# B&R Automation Studio project AutoCon2021 (part 3)

#### AngledMovementFb.st
```iecst
FUNCTION_BLOCK AngledMovementFb
	CASE Internal.state OF
		ANG_INT_OFF:
			IF Execute THEN
				Active := TRUE;
				Internal.ShPos[axPosX] := PosStartX - 0.026;
				Internal.ShPos[axPosY] := PosStartY + 0.026;
				Internal.ShPos[axPosZ] := 0.004;
				Internal.ShPos[axPosRX] := 0.025;
				Internal.ShPos[axPosRY] := 0.025;

				Internal.Fbs.Move6DFb.Controller := ADR(Controller);
				Internal.Fbs.Move6DFb.ShuttleID := ShuttleId;
				Internal.Fbs.Move6DFb.Position := Internal.ShPos;
				Internal.Fbs.Move6DFb.InPlaneVelocity := LinearVel;
				Internal.Fbs.Move6DFb.Acceleration := 10;
				Internal.Fbs.Move6DFb.ShortAxisVelocity[axVel] := LinearVel;
				Internal.Fbs.Move6DFb.ShortAxisVelocity[axVelRx] := ShortAxisRotVel;
				Internal.Fbs.Move6DFb.ShortAxisVelocity[axVelRy] := ShortAxisRotVel;
				Internal.Fbs.Move6DFb.ShortAxisVelocity[axVelRz] := ShortAxisRotVel;

				Internal.Fbs.Move6DFb.Execute := TRUE;

				Internal.state := ANG_INT_MOV_WAIT;
			END_IF
		ANG_INT_MOV_WAIT:
			IF Internal.Fbs.Move6DFb.Done THEN
				Internal.Fbs.Move6DFb.Execute := FALSE;
				Internal.MovementNum := Internal.MovementNum + 1;
				IF Internal.MovementNum >= 11 THEN
					Done := TRUE;
					Internal.state := ANG_INT_DONE;
				ELSE
					Internal.state := ANG_INT_MOV_WAIT + Internal.MovementNum;
				END_IF

			END_IF
		ANG_INT_MOV_1:
			Internal.ShPos[axPosX] := Internal.ShPos[axPosX];
			Internal.ShPos[axPosY] := Internal.ShPos[axPosY] - 0.052;
			Internal.ShPos[axPosRX] := -0.025;
			Internal.ShPos[axPosRY] := 0.025;

			Internal.Fbs.Move6DFb.Position := Internal.ShPos;
			Internal.Fbs.Move6DFb.Execute := TRUE;

			Internal.state := ANG_INT_MOV_WAIT;
		ANG_INT_MOV_2:
			Internal.ShPos[axPosX] := Internal.ShPos[axPosX] + 0.052;
			Internal.ShPos[axPosY] := Internal.ShPos[axPosY];
			Internal.ShPos[axPosRX] := -0.025;
			Internal.ShPos[axPosRY] := -0.025;

			Internal.Fbs.Move6DFb.Position := Internal.ShPos;
			Internal.Fbs.Move6DFb.Execute := TRUE;

			Internal.state := ANG_INT_MOV_WAIT;
		ANG_INT_MOV_3:
			Internal.ShPos[axPosX] := Internal.ShPos[axPosX];
			Internal.ShPos[axPosY] := Internal.ShPos[axPosY] + 0.052;
			Internal.ShPos[axPosRX] := 0.025;
			Internal.ShPos[axPosRY] := -0.025;

			Internal.Fbs.Move6DFb.Position := Internal.ShPos;
			Internal.Fbs.Move6DFb.Execute := TRUE;

			Internal.state := ANG_INT_MOV_WAIT;
		ANG_INT_MOV_4:
			Internal.ShPos[axPosX] := Internal.ShPos[axPosX] - 0.052;
			Internal.ShPos[axPosY] := Internal.ShPos[axPosY];
			Internal.ShPos[axPosRX] := 0.025;
			Internal.ShPos[axPosRY] := 0.025;

			Internal.Fbs.Move6DFb.Position := Internal.ShPos;
			Internal.Fbs.Move6DFb.Execute := TRUE;

			Internal.state := ANG_INT_MOV_WAIT;
		ANG_INT_MOV_5:
			Internal.ShPos[axPosX] := Internal.ShPos[axPosX] + 0.015;
			Internal.ShPos[axPosY] := Internal.ShPos[axPosY] - 0.015;
			Internal.ShPos[axPosRX] := 0.0;
			Internal.ShPos[axPosRY] := 0.0;

			Internal.Fbs.Move6DFb.Position := Internal.ShPos;
			Internal.Fbs.Move6DFb.Execute := TRUE;

			Internal.state := ANG_INT_MOV_WAIT;
		ANG_INT_MOV_6:
			Internal.ShPos[axPosX] := Internal.ShPos[axPosX];
			Internal.ShPos[axPosY] := Internal.ShPos[axPosY] - 0.026;
			Internal.ShPos[axPosRX] := 0.0;
			Internal.ShPos[axPosRY] := 0.0;

			Internal.Fbs.Move6DFb.Position := Internal.ShPos;
			Internal.Fbs.Move6DFb.Execute := TRUE;

			Internal.state := ANG_INT_MOV_WAIT;
		ANG_INT_MOV_7:
			Internal.ShPos[axPosX] := Internal.ShPos[axPosX] + 0.026;
			Internal.ShPos[axPosY] := Internal.ShPos[axPosY];
			Internal.ShPos[axPosRX] := 0.0;
			Internal.ShPos[axPosRY] := 0.0;

			Internal.Fbs.Move6DFb.Position := Internal.ShPos;
			Internal.Fbs.Move6DFb.Execute := TRUE;

			Internal.state := ANG_INT_MOV_WAIT;
		ANG_INT_MOV_8:
			Internal.ShPos[axPosX] := Internal.ShPos[axPosX];
			Internal.ShPos[axPosY] := Internal.ShPos[axPosY] + 0.026;
			Internal.ShPos[axPosRX] := 0.0;
			Internal.ShPos[axPosRY] := 0.0;

			Internal.Fbs.Move6DFb.Position := Internal.ShPos;
			Internal.Fbs.Move6DFb.Execute := TRUE;

			Internal.state := ANG_INT_MOV_WAIT;
		ANG_INT_MOV_9:
			Internal.ShPos[axPosX] := Internal.ShPos[axPosX] - 0.026;
			Internal.ShPos[axPosY] := Internal.ShPos[axPosY];
			Internal.ShPos[axPosRX] := 0.0;
			Internal.ShPos[axPosRY] := 0.0;

			Internal.Fbs.Move6DFb.Position := Internal.ShPos;
			Internal.Fbs.Move6DFb.Execute := TRUE;

			Internal.state := ANG_INT_MOV_WAIT;
		ANG_INT_MOV_10:
			Internal.ShPos[axPosX] := PosStartX;
			Internal.ShPos[axPosY] := PosStartY;
			Internal.ShPos[axPosZ] := 0.002;
			Internal.ShPos[axPosRX] := 0.0;
			Internal.ShPos[axPosRY] := 0.0;

			Internal.Fbs.Move6DFb.Position := Internal.ShPos;
			Internal.Fbs.Move6DFb.Execute := TRUE;

			Internal.state := ANG_INT_MOV_WAIT;

		ANG_INT_DONE:
			IF NOT Execute THEN
				Internal.Fbs.Move6DFb.Execute := FALSE;
				Internal.MovementNum := 0;

				Active := FALSE;
				Done := FALSE;
				Error := FALSE;

				Internal.state := ANG_INT_OFF;
			END_IF
		ANG_INT_ERROR:
			IF NOT Execute THEN
				Internal.Fbs.Move6DFb.Execute := FALSE;
				Internal.MovementNum := 0;

				Active := FALSE;
				Done := FALSE;
				Error := FALSE;

				Internal.state := ANG_INT_OFF;
			END_IF
	END_CASE;
	Internal.Fbs.Move6DFb();
END_FUNCTION_BLOCK
```

#### WobbleMovementFb.st
```iecst
FUNCTION_BLOCK WobbleMovementFb
	//Setup Sun/Planet
	//Run Macro on Virtual
	//Run Wobble Macro on Real
	//When Virtual macro finishes, issue stop command to Real
	//Move6D to real shuttle
	//Exit Sun/Planet
	CASE Internal.state OF
		WOB_INT_OFF:
			IF Execute THEN
				Active := TRUE;

				Internal.Fbs.PlanetCtrlFb.Controller := ADR(Controller);
				Internal.Fbs.PlanetCtrlFb.NumberOfPlanets := 1;
				Internal.Fbs.PlanetCtrlFb.PlanetShuttleID[0] := ShuttleId;
				Internal.Fbs.PlanetCtrlFb.StarShuttleID := VirtShId;
				Internal.Fbs.PlanetCtrlFb.Level := mcACP6D_PLANET_CONNECT;
				Internal.Fbs.PlanetCtrlFb.Execute := TRUE;

				Internal.state := WOB_INT_SETUP_PLANET;
			END_IF
		WOB_INT_SETUP_PLANET:
			IF Internal.Fbs.PlanetCtrlFb.Error THEN
				Internal.state := WOB_INT_ERROR;
			ELSIF Internal.Fbs.PlanetCtrlFb.Done THEN
				Internal.Fbs.PlanetCtrlFb.Execute := FALSE;

				Internal.Fbs.VirtualMacroFb.Controller := ADR(Controller);
				Internal.Fbs.VirtualMacroFb.MacroID := SunMacroID;
				Internal.Fbs.VirtualMacroFb.ShuttleID := VirtShId;
				Internal.Fbs.VirtualMacroFb.Execute := TRUE;

				Internal.Fbs.RealMacroFb.Controller := ADR(Controller);
				Internal.Fbs.RealMacroFb.MacroID := PlanetMacroID;
				Internal.Fbs.RealMacroFb.ShuttleID := ShuttleId;
				Internal.Fbs.RealMacroFb.Execute := TRUE;

				Internal.state := WOB_INT_MACRO_RUN;
			END_IF
		WOB_INT_MACRO_RUN:
			IF Internal.Fbs.RealMacroFb.Error OR Internal.Fbs.VirtualMacroFb.Error THEN
				Internal.state := WOB_INT_ERROR;
			ELSIF Internal.Fbs.VirtualMacroFb.Done THEN
				Internal.Fbs.VirtualMacroFb.Execute := FALSE;
				Internal.Fbs.RealMacroFb.Execute := FALSE;

				Internal.Fbs.StopFb.Controller := ADR(Controller);
				Internal.Fbs.StopFb.ShuttleID := ShuttleId;
				Internal.Fbs.StopFb.Execute := TRUE;

				Internal.state := WOB_INT_STOP;
			END_IF
		WOB_INT_STOP:
			IF Internal.Fbs.StopFb.Error THEN
				Internal.state := WOB_INT_ERROR;
			ELSIF Internal.Fbs.StopFb.Done THEN
				Internal.Fbs.StopFb.Execute := FALSE;

				Internal.Fbs.Move6DFb.Controller := ADR(Controller);
				Internal.Fbs.Move6DFb.ShuttleID := ShuttleId;
				Internal.Fbs.Move6DFb.Position[axPosX] := PosStartX;
				Internal.Fbs.Move6DFb.Position[axPosY] := PosStartY;
				Internal.Fbs.Move6DFb.Position[axPosZ] := 0.002;
				Internal.Fbs.Move6DFb.Position[axPosRX] := 0;
				Internal.Fbs.Move6DFb.Position[axPosRY] := 0;
				Internal.Fbs.Move6DFb.Position[axPosRZ] := 0;
				Internal.Fbs.Move6DFb.InPlaneVelocity := 1;
				Internal.Fbs.Move6DFb.Acceleration := 10;
				Internal.Fbs.Move6DFb.ShortAxisVelocity[axVel] := 1;
				Internal.Fbs.Move6DFb.ShortAxisVelocity[axVelRx] := 0.1;
				Internal.Fbs.Move6DFb.ShortAxisVelocity[axVelRy] := 0.1;
				Internal.Fbs.Move6DFb.ShortAxisVelocity[axVelRz] := 0.1;
				Internal.Fbs.Move6DFb.Execute := TRUE;

				Internal.state := WOB_INT_REORIENT;
			END_IF
		WOB_INT_REORIENT:
			IF Internal.Fbs.Move6DFb.Done THEN
				Internal.Fbs.Move6DFb.Execute := FALSE;

				Internal.Fbs.PlanetCtrlFb.Level := mcACP6D_PLANET_DISCONNECT;
				Internal.Fbs.PlanetCtrlFb.Execute := TRUE;

				Internal.state := WOB_INT_BREAK_PLANET;
			END_IF
		WOB_INT_BREAK_PLANET:
			IF Internal.Fbs.PlanetCtrlFb.Error THEN
				Internal.state := WOB_INT_ERROR;
			ELSIF Internal.Fbs.PlanetCtrlFb.Done THEN
				Internal.Fbs.PlanetCtrlFb.Execute := FALSE;
				Done := TRUE;

				Internal.state := WOB_INT_DONE;
			END_IF
		WOB_INT_DONE:
			IF NOT Execute THEN

				Active := FALSE;
				Done := FALSE;
				Error := FALSE;

				Internal.state := WOB_INT_OFF;
			END_IF
		WOB_INT_ERROR:
			IF NOT Execute THEN
				Internal.Fbs.PlanetCtrlFb.Execute := FALSE;
				Internal.Fbs.RealMacroFb.Execute := FALSE;
				Internal.Fbs.VirtualMacroFb.Execute := FALSE;
				Internal.Fbs.StopFb.Execute := FALSE;
				Internal.Fbs.Move6DFb.Execute := FALSE;

				Active := FALSE;
				Done := FALSE;
				Error := FALSE;

				Internal.state := WOB_INT_OFF;
			END_IF
	END_CASE;
	Internal.Fbs.PlanetCtrlFb();
	Internal.Fbs.RealMacroFb();
	Internal.Fbs.VirtualMacroFb();
	Internal.Fbs.StopFb();
	Internal.Fbs.Move6DFb();
END_FUNCTION_BLOCK
```

#### StationActions.st
```iecst
ACTION SetupStationActions:
	CASE station OF
		ST1:
			FillStationFbs.St1Fb.Execute := TRUE;
			FillStationFbs.St1Fb.Controller := ADR(gMcAcp6DController);
			FillStationFbs.St1Fb.ShuttleId := gShuttleIf[pFillIf.Par.ShuttleIdx].Cfg.ShuttleId;
			FillStationFbs.St1Fb.PosStartX := pFillIf.Cfg.StationPos.X;
			FillStationFbs.St1Fb.PosStartY := pFillIf.Cfg.StationPos.Y;
		ST2:
			FillStationFbs.St2Fb.Controller := ADR(gMcAcp6DController);
			FillStationFbs.St2Fb.MacroID := DINT_TO_USINT(MACRO_FILL_STATION_PROC_2);
			FillStationFbs.St2Fb.ShuttleID := gShuttleIf[pFillIf.Par.ShuttleIdx].Cfg.ShuttleId;
			FillStationFbs.St2Fb.Execute := TRUE;
		ST3:
			FillStationFbs.St3Fb.Controller := ADR(gMcAcp6DController);
			FillStationFbs.St3Fb.PosStartX := pFillIf.Cfg.StationPos.X;
			FillStationFbs.St3Fb.PosStartY := pFillIf.Cfg.StationPos.Y;
			FillStationFbs.St3Fb.PlanetMacroID := DINT_TO_USINT(MACRO_FILL_STATION_PROC_3_WOBBLE);

			FillStationFbs.St3Fb.ShuttleId := gShuttleIf[pFillIf.Par.ShuttleIdx].Cfg.ShuttleId;
			FillStationFbs.St3Fb.VirtShId := 100;
			FillStationFbs.St3Fb.Execute := TRUE;

			CASE macroPatternCounter OF
				0:
					FillStationFbs.St3Fb.SunMacroID := DINT_TO_USINT(MACRO_FILL_STATION_PROC_3_XY);
				1:
					FillStationFbs.St3Fb.SunMacroID := DINT_TO_USINT(MACRO_FILL_STATION_PROC_3_A);
				2:
					FillStationFbs.St3Fb.SunMacroID := DINT_TO_USINT(MACRO_FILL_STATION_PROC_3_B);
			END_CASE;

		ST4:
			FillStationFbs.St4Fb.Controller := ADR(gMcAcp6DController);
			FillStationFbs.St4Fb.MacroID := DINT_TO_USINT(MACRO_FILL_STATION_PROC_4);
			FillStationFbs.St4Fb.ShuttleID := gShuttleIf[pFillIf.Par.ShuttleIdx].Cfg.ShuttleId;
			FillStationFbs.St4Fb.Execute := TRUE;
	END_CASE;
END_ACTION

ACTION CallStationFbs:
	CASE station OF
		ST1:
			FillStationFbs.St1Fb();
		ST2:
			FillStationFbs.St2Fb();
		ST3:
			FillStationFbs.St3Fb();
		ST4:
			FillStationFbs.St4Fb();
	END_CASE;
END_ACTION
```

### Program Logical/Source/ProcessStations/FinishStation (IEC)

#### Cyclic.st - Cyclic code
```iecst
PROGRAM _CYCLIC
	//System operates a batching setup
	//Need two seperate state machines
	//One controls the ouside interface, basically the same as before

	//Second is the internal one, communicates to the external interface as well
	//Process

	//External state machine
	//Waits for a shuttle to be ready
	//When a shuttle is commanded to process
	//Inform the internal state machine a shuttle has arrived
	//Wait for acknowledge, go back to the Wait state

	//FB perhaps?
	//Internal state machine
	//Wait for a shuttle command
	//Send that shuttle to the appropriate destination
		// If the shuttle count is = # of stations, wait for the move to be done
			//Preform the process
		//Else
			//Head back to wait for a more shuttles

	IF NOT gFinishStationIf.Cmd.LocalOverride THEN
		stationPars := gSysPars.FinishStation;
	END_IF

	CASE state OF
		FINISH_OFF: //********************************************************************************Finish station is currently disabled
			IF gFinishStationIf.Cmd.Enable THEN
				stationFbs.BatchProcessFb.Controller := ADR(gMcAcp6DController);
				stationFbs.BatchProcessFb.Enable := TRUE;

				state := FINISH_INIT;
			END_IF
		FINISH_INIT: //********************************************************************************Finish station is initalizing
			IF stationFbs.BatchProcessFb.ReadyForShuttle THEN
				gFinishStationIf.Sts.ReadyForNewShuttle := TRUE;
				gFinishStationIf.Sts.Enabled := TRUE;
				state := FINISH_WAIT_FOR_SHUTTLE;
			END_IF
		FINISH_WAIT_FOR_SHUTTLE: //********************************************************************************Finish station is waiting for a shuttle to be present
			stationFbs.BatchProcessFb.ProcessingTime := stationPars.WaitTime;
			IF NOT gFinishStationIf.Cmd.Enable THEN
				gFinishStationIf.Sts.ReadyForNewShuttle := FALSE;
				gFinishStationIf.Sts.Enabled := FALSE;
				state := FINISH_OFF;
			ELSIF gFinishStationIf.Par.ShuttleIdx <> STATION_IS_EMPTY AND gFinishStationIf.Cmd.Process THEN
				gFinishStationIf.Sts.ReadyForNewShuttle := FALSE;

				stationFbs.BatchProcessFb.ShId := gShuttleIf[gFinishStationIf.Par.ShuttleIdx].Cfg.ShuttleId;
				stationFbs.BatchProcessFb.ProcessShuttle := TRUE;

				state := FINISH_CHECK_BUFFER;
			END_IF
		FINISH_CHECK_BUFFER:
			IF stationFbs.BatchProcessFb.Processsing THEN
				gFinishStationIf.Sts.Processing := TRUE;
				gFinishStationIf.Par.ShuttleIdx := STATION_IS_EMPTY;
				stationFbs.BatchProcessFb.ProcessShuttle := FALSE;

				state := FINISH_FINISHING;
			ELSIF stationFbs.BatchProcessFb.ReadyForShuttle THEN
				gFinishStationIf.Sts.ReadyForNewShuttle := TRUE;
				gFinishStationIf.Par.ShuttleIdx := STATION_IS_EMPTY;
				stationFbs.BatchProcessFb.ProcessShuttle := FALSE;

				state := FINISH_WAIT_FOR_SHUTTLE;
			END_IF
		FINISH_FINISHING: //********************************************************************************Finish station is loading product onto a shuttle
			IF stationFbs.BatchProcessFb.Error THEN
				gFinishStationIf.Sts.Error := TRUE;
				state := FINISH_ERROR;
			ELSIF stationFbs.BatchProcessFb.BatchComplete THEN
				stationFbs.BatchProcessFb.Reset := TRUE;
				gFinishStationIf.Cmd.Process := FALSE;

				gFinishStationIf.Sts.Processing := FALSE;
				FOR i:=0 TO MAX_BATCH_SHUTTLE_COUNT -1 DO
					gShuttleIf[stationFbs.BatchProcessFb.ShuttleIds[i] - 1].Cmd.NextStep := TRUE; //WARNING WARNING THIS WILL ONLY WORK WITH SEQUENTIAL IDS. IF YOU USE ABSOLUTE ID THIS WILL NOT WORK
					gShuttleIf[stationFbs.BatchProcessFb.ShuttleIds[i] - 1].Sts.ProductInfo.Finished := TRUE;
				END_FOR;

				gFinishStationIf.Sts.Done := TRUE;

				state := FINISH_DONE;
			END_IF
		FINISH_DONE: //********************************************************************************Finish station is done with the load process
			IF NOT gFinishStationIf.Cmd.Enable THEN
				gFinishStationIf.Sts.Done := FALSE;
				gFinishStationIf.Sts.Enabled := FALSE;
				gFinishStationIf.Sts.ReadyForNewShuttle := FALSE;
				stationFbs.BatchProcessFb.Enable := FALSE;

				state := FINISH_OFF;
			ELSIF NOT gFinishStationIf.Cmd.Process AND stationFbs.BatchProcessFb.ReadyForShuttle THEN
				gFinishStationIf.Par.ShuttleIdx := STATION_IS_EMPTY;
				gFinishStationIf.Sts.Done := FALSE;
				gFinishStationIf.Sts.ReadyForNewShuttle := FALSE;
				gFinishStationIf.Sts.ReadyForNewShuttle := TRUE;

				state := FINISH_WAIT_FOR_SHUTTLE;
			END_IF

		FINISH_ERROR: //********************************************************************************Finish station had an error
			IF gFinishStationIf.Cmd.Reset THEN
				gFinishStationIf.Cmd.Reset := FALSE;

				gFinishStationIf.Sts.Done := FALSE;
				gFinishStationIf.Sts.Enabled := FALSE;
				gFinishStationIf.Sts.Error := FALSE;
				gFinishStationIf.Sts.Processing := FALSE;
				gFinishStationIf.Sts.ReadyForNewShuttle := FALSE;

				gFinishStationIf.Par.ShuttleIdx := STATION_IS_EMPTY;
				IF gFinishStationIf.Cmd.Enable THEN
					state := FINISH_INIT;
				ELSE
					state := FINISH_OFF;
				END_IF
			END_IF
	END_CASE;

	 stationFbs.BatchProcessFb();
END_PROGRAM
```

#### Init.st - Init code
```iecst
PROGRAM _INIT
	gFinishStationIf.Par.ShuttleIdx := STATION_IS_EMPTY;
	//Define station configuration values
	gFinishStationIf.Cfg.StationPos.X := 0.9;
	gFinishStationIf.Cfg.StationPos.Y := 0.9;

	stationFbs.BatchProcessFb.Positions[0].X := 0.9;
	stationFbs.BatchProcessFb.Positions[0].Y := 1.26;
	stationFbs.BatchProcessFb.Positions[1].X := 0.9;
	stationFbs.BatchProcessFb.Positions[1].Y := 1.14;

	gSysPars.FinishStation.WaitTime := T#1s;
END_PROGRAM
```

#### Types.typ - Local data types
```iecst
TYPE
	FinishStationStateEnum :
		(
		FINISH_OFF, (*Finish station is currently disabled*)
		FINISH_INIT, (*Finish station is initalizing*)
		FINISH_WAIT_FOR_SHUTTLE, (*Finish station is waiting for a shuttle to be present*)
		FINISH_CHECK_BUFFER, (*Finish station is Checking on the buffer status *)
		FINISH_FINISHING, (*Finish station is preforming the batch finishing process on the shuttles*)
		FINISH_DONE, (*Finish station is done with the finish process*)
		FINISH_ERROR (*Finish station had an error*)
		);
	FinishStationFbTyp : 	STRUCT
		BatchProcessFb : BatchProcess6DFb;
	END_STRUCT;
END_TYPE
```

#### Variables.var - Local variables
```iecst
VAR
	state : FinishStationStateEnum;
	stationFbs : FinishStationFbTyp;
	stationPars : FinishStationParsTyp;
	i : INT;
END_VAR
```

#### LocalFunctionsTyp.typ - Local data types
```iecst
TYPE
	BatchProcess6DInternalTyp : 	STRUCT
		State : BatchProcess6DStateEnum;
		currentShuttleCount : USINT;
		Fbs : BatchProcess6DFbsTyp;
	END_STRUCT;
	BatchProcess6DStateEnum :
		(
		BATCH_OFF,
		BATCH_INIT,
		BATCH_WAIT_SHUTTLE,
		BATCH_MOVE_SHUTTLE,
		BATCH_PREFORM_OPERATION,
		BATCH_DONE,
		BATCH_RESET,
		BATCH_ERROR
		);
	BatchProcess6DFbsTyp : 	STRUCT
		MoveInPlaneFb : MC_BR_MoveInPlane_Acp6D;
		WaitTimer : TON;
	END_STRUCT;
END_TYPE
```

#### LocalFunctions.fun
```iecst
{REDUND_ERROR} FUNCTION_BLOCK BatchProcess6DFb (*TODO: Add your comment here*) (*$GROUP=User,$CAT=User,$GROUPICON=User.png,$CATICON=User.png*)
	VAR_INPUT
		Controller : REFERENCE TO McAcp6DControllerType;
		Enable : BOOL;
		Reset : BOOL;
		ProcessingTime : TIME;
		Positions : {REDUND_UNREPLICABLE} ARRAY[0..MAX_BATCH_SHUTTLE_COUNT_ARRAY] OF StationPositionTyp;
		ProcessShuttle : BOOL;
		ShId : USINT;
	END_VAR
	VAR_OUTPUT
		Error : BOOL;
		StatusID : DINT;
		ReadyForShuttle : BOOL;
		Processsing : BOOL;
		BatchComplete : BOOL;
		ShuttleIds : ARRAY[0..MAX_BATCH_SHUTTLE_COUNT_ARRAY] OF USINT;
	END_VAR
	VAR
		Internal : BatchProcess6DInternalTyp;
	END_VAR
END_FUNCTION_BLOCK
```

### Program Logical/Source/ProcessStations/RejectStation

#### Types.typ
```iecst
TYPE
	RejectStationStateEnum :
		(
		REJECT_OFF, (*Reject station is currently disabled*)
		REJECT_INIT, (*Reject station is initalizing*)
		REJECT_WAIT_FOR_SHUTTLE, (*Reject station is waiting for a shuttle to be present*)
		REJECT_REJECTING, (*Reject station is rejecting product from the shuttle*)
		REJECT_DONE, (*Reject station is done with the weigh process*)
		REJECT_ERROR (*Reject station had an error*)
		);
	RejectStationFbTyp : 	STRUCT
		RejectTimerFb : TON;
	END_STRUCT;
END_TYPE
```

#### Variables.var
```iecst
VAR
	state : RejectStationStateEnum;
	stFbs : {REDUND_UNREPLICABLE} RejectStationFbTyp;
	stationPars : {REDUND_UNREPLICABLE} RejectStationParsTyp;
END_VAR
```

#### Cyclic.st
```iecst
PROGRAM _CYCLIC
	IF NOT gRejectStationIf.Cmd.LocalOverride THEN
		stationPars := gSysPars.RejectStation;
	END_IF
	CASE state OF
		REJECT_OFF: //********************************************************************************Reject station is currently disabled
			IF gRejectStationIf.Cmd.Enable THEN
				state := REJECT_INIT;
			END_IF
		REJECT_INIT: //********************************************************************************Reject station is initalizing
			gRejectStationIf.Sts.ReadyForNewShuttle := TRUE;
			gRejectStationIf.Sts.Enabled := TRUE;
			state := REJECT_WAIT_FOR_SHUTTLE;
		REJECT_WAIT_FOR_SHUTTLE: //********************************************************************************Reject station is waiting for a shuttle to be present
			IF NOT gRejectStationIf.Cmd.Enable THEN
				gRejectStationIf.Sts.ReadyForNewShuttle := FALSE;
				gRejectStationIf.Sts.Enabled := FALSE;
				state := REJECT_OFF;
			ELSIF gRejectStationIf.Par.ShuttleIdx <> STATION_IS_EMPTY AND gRejectStationIf.Cmd.Process THEN
				gRejectStationIf.Sts.ReadyForNewShuttle := FALSE;
				gRejectStationIf.Sts.Processing := TRUE;

				stFbs.RejectTimerFb.IN := TRUE;
				stFbs.RejectTimerFb.PT := stationPars.WaitTime;

				state := REJECT_REJECTING;
			END_IF
		REJECT_REJECTING: //********************************************************************************Reject station is weighing product onto a shuttle
			IF stFbs.RejectTimerFb.Q THEN
				stFbs.RejectTimerFb.IN := FALSE;

				gRejectStationIf.Sts.Processing := FALSE;
				gShuttleIf[gRejectStationIf.Par.ShuttleIdx].Sts.ProductInfo.Loaded := FALSE;
				gShuttleIf[gRejectStationIf.Par.ShuttleIdx].Cmd.NextStep := TRUE;
				gRejectStationIf.Sts.Done := TRUE;

				state := REJECT_DONE;
			END_IF
		REJECT_DONE: //********************************************************************************Reject station is done with the weigh process
			IF NOT gRejectStationIf.Cmd.Enable THEN
				gRejectStationIf.Sts.Done := FALSE;
				gRejectStationIf.Sts.Enabled := FALSE;
				gRejectStationIf.Sts.ReadyForNewShuttle := FALSE;
				state := REJECT_OFF;
			ELSIF NOT gRejectStationIf.Cmd.Process THEN
				gRejectStationIf.Par.ShuttleIdx := STATION_IS_EMPTY;
				gRejectStationIf.Sts.Done := FALSE;
				gRejectStationIf.Sts.ReadyForNewShuttle := TRUE;

				state := REJECT_WAIT_FOR_SHUTTLE;
			END_IF

		REJECT_ERROR: //********************************************************************************Reject station had an error
			IF gRejectStationIf.Cmd.Reset THEN
				gRejectStationIf.Cmd.Reset := FALSE;

				gRejectStationIf.Sts.Done := FALSE;
				gRejectStationIf.Sts.Enabled := FALSE;
				gRejectStationIf.Sts.Error := FALSE;
				gRejectStationIf.Sts.Processing := FALSE;
				gRejectStationIf.Sts.ReadyForNewShuttle := FALSE;

				stFbs.RejectTimerFb.IN := FALSE;

				gRejectStationIf.Par.ShuttleIdx := STATION_IS_EMPTY;
				IF gRejectStationIf.Cmd.Enable THEN
					state := REJECT_INIT;
				ELSE
					state := REJECT_OFF;
				END_IF
			END_IF
	END_CASE;

	stFbs.RejectTimerFb();

END_PROGRAM
```

#### Init.st
```iecst
PROGRAM _INIT
	gRejectStationIf.Par.ShuttleIdx := STATION_IS_EMPTY;

	gRejectStationIf.Cfg.StationPos.X := 0.78;
	gRejectStationIf.Cfg.StationPos.Y := 0.54;
	//Define station configuration values
	gSysPars.RejectStation.WaitTime := T#2s;

	gSysPars.RejectStation.FailPercentage := 90;
END_PROGRAM
```

### Program Logical/Source/ProcessStations/WeighStation

#### Types.typ
```iecst
TYPE
	WeighStationStateEnum :
		(
		WEIGH_OFF, (*Weigh station is currently disabled*)
		WEIGH_INIT, (*Weigh station is initalizing*)
		WEIGH_WAIT_FOR_SHUTTLE, (*Weigh station is waiting for a shuttle to be present*)
		WEIGH_LAND, (*Weigh station is landing a shuttle*)
		WEIGH_TAKEOFF, (*Weigh station is taking off a shuttle*)
		WEIGH_WEIGHING, (*Weigh station is weighing product onto a shuttle*)
		WEIGH_DONE, (*Weigh station is done with the weigh process*)
		WEIGH_ERROR (*Weigh station had an error*)
		);
	WeighStationFbTyp : 	STRUCT
		WeighTimerFb : TON;
		LevitationCtrlFb : MC_BR_LevitationCtrl_Acp6D;
	END_STRUCT;
END_TYPE
```

#### Variables.var
```iecst
VAR
	state : WeighStationStateEnum;
	stFbs : WeighStationFbTyp;
	pWeighIf : REFERENCE TO StationIfTyp;
	taskName : STRING[80];
	stationPars : REFERENCE TO WeighStationParsTyp;
	i : INT;
	lastRecordedWeight : DINT;
	lastRecordedWeightHMI : REAL;
END_VAR
```

#### Cyclic.st
```iecst
PROGRAM _CYCLIC

	CASE state OF
		WEIGH_OFF: //********************************************************************************Weigh station is currently disabled
			IF pWeighIf.Cmd.Enable THEN
				state := WEIGH_INIT;
			END_IF
		WEIGH_INIT: //********************************************************************************Weigh station is initalizing
			pWeighIf.Sts.ReadyForNewShuttle := TRUE;
			pWeighIf.Sts.Enabled := TRUE;
			state := WEIGH_WAIT_FOR_SHUTTLE;
		WEIGH_WAIT_FOR_SHUTTLE: //********************************************************************************Weigh station is waiting for a shuttle to be present
			IF NOT pWeighIf.Cmd.Enable THEN
				pWeighIf.Sts.ReadyForNewShuttle := FALSE;
				pWeighIf.Sts.Enabled := FALSE;
				state := WEIGH_OFF;
			ELSIF pWeighIf.Par.ShuttleIdx <> STATION_IS_EMPTY AND pWeighIf.Cmd.Process THEN
				pWeighIf.Sts.ReadyForNewShuttle := FALSE;

				state := WEIGH_LAND;
			END_IF
		WEIGH_LAND: //********************************************************************************Weigh station is landing a shuttle
			stFbs.LevitationCtrlFb.Controller := ADR(gMcAcp6DController);
			stFbs.LevitationCtrlFb.ShuttleID := gShuttleIf[pWeighIf.Par.ShuttleIdx].Cfg.ShuttleId;
			stFbs.LevitationCtrlFb.Level := mcACP6D_LEVEL_LAND;
			stFbs.LevitationCtrlFb.Execute := TRUE;

			IF stFbs.LevitationCtrlFb.Error THEN
				state := WEIGH_ERROR;
			ELSIF stFbs.LevitationCtrlFb.Done THEN
				stFbs.LevitationCtrlFb.Execute := FALSE;

				state := WEIGH_TAKEOFF;
			END_IF
		WEIGH_TAKEOFF: //********************************************************************************Weigh station is taking off a shuttle
			stFbs.LevitationCtrlFb.Controller := ADR(gMcAcp6DController);
			stFbs.LevitationCtrlFb.ShuttleID := gShuttleIf[pWeighIf.Par.ShuttleIdx].Cfg.ShuttleId;
			stFbs.LevitationCtrlFb.Level := mcACP6D_LEVEL_LEVITATE;
			stFbs.LevitationCtrlFb.Execute := TRUE;

			IF stFbs.LevitationCtrlFb.Error THEN
				state := WEIGH_ERROR;
			ELSIF stFbs.LevitationCtrlFb.Done THEN
				stFbs.LevitationCtrlFb.Execute := FALSE;

				stFbs.WeighTimerFb.IN := TRUE;
				pWeighIf.Sts.Processing := TRUE;
				stFbs.WeighTimerFb.PT := stationPars.WaitTime;

				state := WEIGH_WEIGHING;
			END_IF
		WEIGH_WEIGHING: //********************************************************************************Weigh station is weighing product onto a shuttle
			IF stFbs.WeighTimerFb.Q THEN
				stFbs.WeighTimerFb.IN := FALSE;

				lastRecordedWeight := RandValueDINT(stationPars.MinWeight,stationPars.MaxWeight);
				lastRecordedWeightHMI := DINT_TO_REAL(lastRecordedWeight) / 10.0;
				gShuttleIf[pWeighIf.Par.ShuttleIdx].Sts.ProductInfo.Weight := DINT_TO_REAL(lastRecordedWeight) / 10.0;

				pWeighIf.Sts.Processing := FALSE;
				gShuttleIf[pWeighIf.Par.ShuttleIdx].Cmd.NextStep := TRUE;
				pWeighIf.Sts.Done := TRUE;

				state := WEIGH_DONE;
			END_IF
		WEIGH_DONE: //********************************************************************************Weigh station is done with the weigh process
			IF NOT pWeighIf.Cmd.Enable THEN
				pWeighIf.Sts.Done := FALSE;
				pWeighIf.Sts.Enabled := FALSE;
				pWeighIf.Sts.ReadyForNewShuttle := FALSE;
				state := WEIGH_OFF;
			ELSIF NOT pWeighIf.Cmd.Process THEN
				pWeighIf.Par.ShuttleIdx := STATION_IS_EMPTY;
				pWeighIf.Sts.Done := FALSE;
				pWeighIf.Sts.ReadyForNewShuttle := FALSE;
				pWeighIf.Sts.ReadyForNewShuttle := TRUE;

				state := WEIGH_WAIT_FOR_SHUTTLE;
			END_IF

		WEIGH_ERROR: //********************************************************************************Weigh station had an error
			IF pWeighIf.Cmd.Reset THEN
				pWeighIf.Cmd.Reset := FALSE;

				pWeighIf.Sts.Done := FALSE;
				pWeighIf.Sts.Enabled := FALSE;
				pWeighIf.Sts.Error := FALSE;
				pWeighIf.Sts.Processing := FALSE;
				pWeighIf.Sts.ReadyForNewShuttle := FALSE;

				stFbs.WeighTimerFb.IN := FALSE;
				stFbs.LevitationCtrlFb.Execute := FALSE;

				pWeighIf.Par.ShuttleIdx := STATION_IS_EMPTY;
				IF pWeighIf.Cmd.Enable THEN
					state := WEIGH_INIT;
				ELSE
					state := WEIGH_OFF;
				END_IF
			END_IF
	END_CASE;

	stFbs.WeighTimerFb();
	stFbs.LevitationCtrlFb();

END_PROGRAM
```

#### Init.st
```iecst
PROGRAM _INIT
	ST_name(0,ADR(taskName),0);

	IF taskName = 'WeighSt1' THEN
		pWeighIf ACCESS ADR(gWeighStationIf[0]);
		stationPars ACCESS ADR(gSysPars.WeighStations[0]);

		pWeighIf.Par.ShuttleIdx := STATION_IS_EMPTY;
		pWeighIf.Cfg.StationPos.X := 1.14;
		pWeighIf.Cfg.StationPos.Y := 0.9;
	ELSIF taskName = 'WeighSt2' THEN
		pWeighIf ACCESS ADR(gWeighStationIf[1]);
		stationPars ACCESS ADR(gSysPars.WeighStations[1]);

		pWeighIf.Par.ShuttleIdx := STATION_IS_EMPTY;
		pWeighIf.Cfg.StationPos.X := 1.02;
		pWeighIf.Cfg.StationPos.Y := 0.9;
	END_IF
	//Define station configuration values

	FOR i:=0 TO MAX_WEIGH_STATIONS - 1 DO
		gSysPars.WeighStations[i].WaitTime := T#300ms;
		gSysPars.WeighStations[i].MinWeight := 4300;
		gSysPars.WeighStations[i].MaxWeight := 4320;
	END_FOR;
END_PROGRAM
```

### Package Logical/Source/Main - Package that contains the main entry point to the machine

### Program Logical/Source/Main/Main (IEC)

#### Cyclic.st - Cyclic code
```iecst
PROGRAM _CYCLIC
	IF gAcp6DCtrlIf.Status.Error THEN
		state := MAIN_ERROR;
	END_IF

	CASE state OF
		MAIN_OFF: //******************************************************************************** Main Off State
			IF gMainIf.Cmd.Power THEN
				gAcp6DCtrlIf.Cmd.Power := TRUE;

				state := MAIN_INIT;
			END_IF
		MAIN_INIT: //******************************************************************************** Main Initializing State
			IF gAcp6DCtrlIf.Status.PowerOn AND gAcp6DCtrlIf.Status.Ready THEN
				gMainIf.Status.PowerOn := TRUE;
				g6DRecoveryIf.Cmd.Recover := TRUE;

				state := MAIN_RECOVERING;
			ELSIF NOT gMainIf.Cmd.Power THEN
				gAcp6DCtrlIf.Cmd.Power := FALSE;
				state := MAIN_OFF;
			END_IF
		MAIN_RECOVERING: //******************************************************************************** Main Recovery State
			IF g6DRecoveryIf.Sts.ReadyToStartProc THEN
				g6DRecoveryIf.Cmd.Recover := FALSE;

				state := MAIN_READY;
			END_IF
		MAIN_READY://******************************************************************************** Main Ready State
			IF gMainIf.Cmd.Start THEN
				gLoadStationIf.Cmd.Enable := TRUE;
				gUnloadStationIf.Cmd.Enable := TRUE;
				gPrintStationIf.Cmd.Enable := TRUE;
				gDoseStationsIf[0].Cmd.Enable := TRUE;
				gDoseStationsIf[1].Cmd.Enable := TRUE;
				gTampStationIf.Cmd.Enable := TRUE;
				gProcessInfoIf.Cmd.Enable := TRUE;
				CmdShEnable(TRUE, ADR(gShuttleIf), gMainIf.Cfg.ShuttleCount);

				state := MAIN_STARTING;
			ELSIF NOT gMainIf.Cmd.Power THEN
				gMainIf.Status.PowerOn := FALSE;
				gAcp6DCtrlIf.Cmd.Power := FALSE;
				state := MAIN_OFF;
			END_IF
		MAIN_STARTING://******************************************************************************** Main Starting State
			IF gLoadStationIf.Status.Enabled
				AND gUnloadStationIf.Status.Enabled
				AND gPrintStationIf.Status.Enabled
				AND gDoseStationsIf[0].Status.Enabled
				AND gDoseStationsIf[1].Status.Enabled
				AND gTampStationIf.Status.Enabled
				AND gProcessInfoIf.Sts.Enabled THEN

				gMainIf.Cmd.Start := FALSE;
				state := MAIN_RUNNING;
			END_IF

		MAIN_RUNNING: //******************************************************************************** Main Running State
			IF gMainIf.Cmd.Stop THEN
				gLoadStationIf.Cmd.Enable := FALSE;
				gUnloadStationIf.Cmd.Enable := FALSE;
				gPrintStationIf.Cmd.Enable := FALSE;
				gDoseStationsIf[0].Cmd.Enable := FALSE;
				gDoseStationsIf[1].Cmd.Enable := FALSE;
				gTampStationIf.Cmd.Enable := FALSE;
				gProcessInfoIf.Cmd.Enable := FALSE;

				state := MAIN_STOPPING;
			END_IF
		MAIN_STOPPING: //******************************************************************************** Main Stopping State
			IF NOT gLoadStationIf.Status.Enabled
				AND NOT gUnloadStationIf.Status.Enabled
				AND NOT gPrintStationIf.Status.Enabled
				AND NOT gDoseStationsIf[0].Status.Enabled
				AND NOT gDoseStationsIf[1].Status.Enabled
				AND NOT gTampStationIf.Status.Enabled
				AND NOT gProcessInfoIf.Sts.Enabled THEN

				gMainIf.Cmd.Stop := FALSE;

				FOR i:=0 TO gMainIf.Cfg.ShuttleCount - 1 DO
					gShuttleIf[i].Status.Recovered := FALSE;
				END_FOR;

				state := MAIN_READY;
			END_IF

		MAIN_ERROR: //******************************************************************************** Main Error State
			IF gMainIf.Cmd.Reset THEN
				gMainIf.Cmd.Reset := FALSE;
				gAcp6DCtrlIf.Cmd.ErrorReset := TRUE;

				state := MAIN_OFF;
			END_IF
	END_CASE;

END_PROGRAM
```

#### Init.st - Init code
```iecst
PROGRAM _INIT
	gMainIf.Cfg.ShuttleCount := 8;

	//Used to initialize the shuttle indecies.
	FOR i:=0 TO gMainIf.Cfg.ShuttleCount-1 DO
		gShuttleIf[i].Cfg.ShuttleId := i + 1;
	END_FOR;

END_PROGRAM
```

#### Types.typ - Local data types
```iecst
TYPE
	MainStatesEnum :
		(
		MAIN_OFF,
		MAIN_INIT,
		MAIN_RECOVERING,
		MAIN_READY,
		MAIN_STARTING,
		MAIN_RUNNING,
		MAIN_STOPPING,
		MAIN_ERROR
		);
END_TYPE
```

#### Variables.var - Local variables
```iecst
VAR
	i : USINT; (*Loop index*)
	state : MainStatesEnum; (*State of system*)
END_VAR
```

#### LocalFunctions.typ
```iecst
TYPE
	CmdShEnableInternalTyp : 	STRUCT
		EnableCheck : BOOL;
		i : USINT;
	END_STRUCT;
END_TYPE
```

#### LocalFunctions.fun
```iecst
{REDUND_ERROR} FUNCTION CmdShEnable : BOOL (*Provides interface to group enable command for all shuttles*) (*$GROUP=User,$CAT=User,$GROUPICON=User.png,$CATICON=User.png*)
	VAR_INPUT
		Enable : BOOL;
		ShIfs : REFERENCE TO ARRAY[0..MAX_SHUTTLE_COUNT_ARRAY] OF gShuttleIfTyp;
		ShCount : USINT;
	END_VAR
	VAR
		Internal : CmdShEnableInternalTyp;
	END_VAR
END_FUNCTION
```

#### CmdShEnable.st
```iecst
(* Provides interface to group enable command for all shuttles *)
FUNCTION CmdShEnable
	Internal.EnableCheck := TRUE;
	FOR Internal.i:=0 TO ShCount-1 DO
		ShIfs[Internal.i].Cmd.Enable := Enable;
	END_FOR;
	CmdShEnable := Internal.EnableCheck;
END_FUNCTION
```

#### CmdShStop.st - not listed in the package file held
```iecst
(* Provides interface to group enable command for all shuttles *)
FUNCTION CmdShStop
	FOR Internal.i:=0 TO ShCount-1 DO
		ShIfs[Internal.i].Cmd.Stop := TRUE;
	END_FOR;
	CmdShStop := Internal.StopCheck;
END_FUNCTION
```

### Package Logical/Source/6DCtrl - Package containing the main logic for controlling the 6D system as a whole

### Acp6DGlobalVars.var
```iecst
VAR CONSTANT
	MAX_MACRO_COUNT : USINT := 63;
	MAX_MACRO_COUNT_ARRAY : USINT := MAX_MACRO_COUNT-1;
END_VAR
VAR
	gMacroLoadIf : gMacroLoadIfTYp;
END_VAR
```

### Acp6DTypes.typ
```iecst
(*Datatypes for the Load Macro Interface*)

TYPE
	gMacroLoadIfTYp : 	STRUCT
		Cmd : gMacroLoadIfCmdTyp;
		Par : gMacroLoadIfParTyp;
		Status : gMacroLoadIfStatusTyp;
	END_STRUCT;
	gMacroLoadIfCmdTyp : 	STRUCT
		LoadAll : BOOL; (*Command to load all macros*)
		Clear : BOOL; (*Command to clear a singular macro*)
		LoadSingle : BOOL; (*Commadn to load a singular macro*)
		Reset : BOOL; (*Command to reset the macro load interface. Also resets the "AllMacroLoaded" status*)
	END_STRUCT;
	MacroParTyp : 	STRUCT
		Load : BOOL; (*Flag To denote that we should load the macro*)
		MacroFileName : STRING[80]; (*XML File Name of the Macro to load*)
		MacroID : USINT; (*MacroID of the associated macro*)
	END_STRUCT;
	gMacroLoadIfParTyp : 	STRUCT
		FileDevice : STRING[80]; (*FileDevice to find the macro *)
		MacroList : ARRAY[0..MAX_MACRO_COUNT_ARRAY]OF MacroParTyp; (*List of macros to load*)
		SingleMacroLoad : MacroParTyp; (*Parameter to load a singular macro*)
	END_STRUCT;
	gMacroLoadIfStatusTyp : 	STRUCT
		AllMacrosLoaded : BOOL;
		Loading : BOOL;
		CurrentMacro : USINT;
		CmdDone : BOOL;
		Error : BOOL;
		MacroIDError : USINT;
	END_STRUCT;
END_TYPE
```

### Program Logical/Source/6DCtrl/6DCtrl (IEC)

#### Types.typ
```iecst
TYPE
	Acp6DStateEnum :
		( (*6D Control States*)
		ACP6D_RESET, (*Reset the 6D controller state*)
		ACP6D_POWER_OFF, (*System Power Off state*)
		ACP6D_INACTIVE, (*System inactive state*)
		ACP6D_POWER_ON, (*Powering on the system state*)
		ACP6D_WAIT_ACTIVATION, (*waiting for activation (needed for autoID)*)
		ACP6D_INIT_MACRO, (*Waiting for the initalization of the macros to be done*)
		ACP6D_READY, (*System Ready for operation*)
		ACP6D_ERROR := 255 (*System in an error state*)
		);
	Sys6DCtrlFbTyp : 	STRUCT
		AutoRefreshFB : MC_BR_AutoRefresh_Acp6D; (*FB that auto refreshes the 6D data*)
		PowerOnFb : MC_BR_SysPowerOn_Acp6D; (*FB to power on the 6D controller/system*)
		PowerOffFb : MC_BR_SysPowerOff_Acp6D; (*FB to power off the 6D controller/system*)
		SysReadStateFb : MC_BR_SysReadState_Acp6D; (*FB to read the state of the 6D controller*)
		ShReadPositionFb : ARRAY[0..MAX_SHUTTLE_COUNT_ARRAY]OF MC_BR_ShReadPosition_Acp6D; (*FB(s) to read the position of the shuttles*)
		ShReadForceFb : ARRAY[0..MAX_SHUTTLE_COUNT_ARRAY]OF MC_BR_ShReadForce_Acp6D; (*FB(s) to read the force acting on the shuttle*)
		ShReadState : ARRAY[0..MAX_SHUTTLE_COUNT_ARRAY]OF MC_BR_ShReadState_Acp6D; (*FB(s) to read the states of the shuttles*)
		GetErrorCodesFb : MC_BR_GetErrorCode_Acp6D; (*FB to read the error codes on the 6D controller*)
	END_STRUCT;
END_TYPE
```

#### Variables.var
```iecst
VAR
	Fbs : Sys6DCtrlFbTyp; (*Function Blocks to Ctrl 6D system*)
	state : Acp6DStateEnum; (*Acp6d state*)
	i : USINT; (*Loop index counter*)
END_VAR
```

#### Cyclic.st
```iecst
PROGRAM _CYCLIC

	IF((Fbs.SysReadStateFb.Valid AND Fbs.SysReadStateFb.State = mcACP6D_STATE_ERROR) AND (state <> ACP6D_ERROR))THEN
		state := ACP6D_ERROR;
	END_IF;

	CASE state OF
		ACP6D_RESET: 	//******************************************************************************** 6D Reset State
			IF(Fbs.SysReadStateFb.Valid AND (Fbs.SysReadStateFb.State = mcACP6D_STATE_INACTIVE))THEN
				state := ACP6D_INACTIVE;
			ELSIF(Fbs.SysReadStateFb.State = mcACP6D_STATE_OPERATION)THEN
				state := ACP6D_POWER_OFF;
			END_IF;

		ACP6D_POWER_OFF: 	//******************************************************************************** 6D Power off commanding State
			Fbs.PowerOffFb.Execute := TRUE;
			IF(Fbs.PowerOffFb.Acknowledge AND (Fbs.SysReadStateFb.Valid AND Fbs.SysReadStateFb.State = mcACP6D_STATE_INACTIVE))THEN
				gAcp6DCtrlIf.Status.PowerOn := FALSE;
				Fbs.PowerOffFb.Execute 	:= FALSE;
				state := ACP6D_INACTIVE;
			ELSIF(Fbs.PowerOffFb.Error)THEN
				Fbs.PowerOffFb.Execute 	:= FALSE;
				gAcp6DCtrlIf.Status.ErrorID := Fbs.PowerOffFb.ErrorID;
				state := ACP6D_ERROR;
			END_IF;

		ACP6D_INACTIVE:	 	//******************************************************************************** 6D Inactive/Power Off state
			IF(gAcp6DCtrlIf.Cmd.Power)THEN
				Fbs.PowerOnFb.Execute := TRUE;
				//MpAuditCustomEvent(gAuditTrail,"INFO","Acp6DSys","Power On Command Issued");
				state := ACP6D_POWER_ON;
			END_IF;

		ACP6D_POWER_ON: 	//******************************************************************************** 6D Power on Commanding State
			IF Fbs.PowerOnFb.Error THEN
				gAcp6DCtrlIf.Status.ErrorID := Fbs.PowerOnFb.ErrorID;
				state := ACP6D_ERROR;
			ELSIF(Fbs.PowerOnFb.Acknowledge AND (Fbs.SysReadStateFb.Valid AND (Fbs.SysReadStateFb.State > mcACP6D_STATE_INACTIVE)))THEN
				//MpAuditCustomEvent(gAuditTrail,"INFO","Acp6DSys","Powered On");
				Fbs.PowerOnFb.Execute := FALSE;
				state := ACP6D_WAIT_ACTIVATION;
			END_IF;

			//Necessary state when using Absolute ID.
		ACP6D_WAIT_ACTIVATION: 	//******************************************************************************** 6D Waiting for Activation of Shuttles State
			IF(Fbs.SysReadStateFb.Valid)THEN
				IF(Fbs.SysReadStateFb.State = mcACP6D_STATE_OPERATION)THEN
					gAcp6DCtrlIf.Status.PowerOn := TRUE;
					state := ACP6D_INIT_MACRO;
				ELSIF(Fbs.SysReadStateFb.State = mcACP6D_STATE_INACTIVE)THEN
					state := ACP6D_INACTIVE; // Error during Activating state; Can happen in Absolute ID mode.
					gAcp6DCtrlIf.Cmd.Power := FALSE;
				END_IF;
			END_IF;
		ACP6D_INIT_MACRO: 	//******************************************************************************** 6D Wait for Macro initilization State
			IF gMacroLoadIf.Status.AllMacrosLoaded THEN
				gMacroLoadIf.Cmd.LoadAll := FALSE;
				state := ACP6D_READY;
			ELSE
				gMacroLoadIf.Cmd.LoadAll := TRUE;
			END_IF

		ACP6D_READY: 	//******************************************************************************** 6D Ready/Running State
			IF(NOT gAcp6DCtrlIf.Cmd.Power)THEN
				gMacroLoadIf.Cmd.Reset := TRUE;
				state := ACP6D_POWER_OFF;
			END_IF;

		ACP6D_ERROR: 	//******************************************************************************** 6D Error State
			gAcp6DCtrlIf.Status.PowerOn := FALSE;
			IF(gAcp6DCtrlIf.Cmd.ErrorReset)THEN
				IF(Fbs.SysReadStateFb.State<>mcACP6D_STATE_ERROR)THEN
					gAcp6DCtrlIf.Cmd.ErrorReset := FALSE;
					state := ACP6D_RESET;
				ELSE
					Fbs.PowerOffFb.Execute := TRUE;	 // Reset error with power off.
					IF(Fbs.PowerOffFb.Acknowledge)THEN
						gMacroLoadIf.Cmd.Reset := TRUE;
						Fbs.PowerOffFb.Execute 	:= FALSE;
					ELSIF(Fbs.PowerOffFb.Error)THEN
						gAcp6DCtrlIf.Cmd.ErrorReset := FALSE;
						Fbs.PowerOffFb.Execute 	:= FALSE;
						gAcp6DCtrlIf.Status.ErrorID := Fbs.PowerOffFb.ErrorID;
						state := ACP6D_ERROR;
					END_IF;
				END_IF;
			END_IF;
	END_CASE;

	FOR i:=0 TO gMainIf.Cfg.ShuttleCount - 1 DO
		Fbs.ShReadPositionFb[i].Controller := ADR(gMcAcp6DController);
		Fbs.ShReadPositionFb[i].Enable := TRUE;
		Fbs.ShReadPositionFb[i].ShuttleID := gShuttleIf[i].Cfg.ShuttleId;
		Fbs.ShReadPositionFb[i]();

		Fbs.ShReadForceFb[i].Controller := ADR(gMcAcp6DController);
		Fbs.ShReadForceFb[i].Enable := TRUE;
		Fbs.ShReadForceFb[i].ShuttleID := gShuttleIf[i].Cfg.ShuttleId;
		Fbs.ShReadForceFb[i]();

		Fbs.ShReadState[i].Controller := ADR(gMcAcp6DController);
		Fbs.ShReadState[i].Enable := TRUE;
		Fbs.ShReadState[i].ShuttleID := gShuttleIf[i].Cfg.ShuttleId;
		Fbs.ShReadState[i]();

		gShuttleIf[i].Status.ShuttleInfo.Force.Value := Fbs.ShReadForceFb[i].ForceInfo;
		gShuttleIf[i].Status.ShuttleInfo.Force.Valid := Fbs.ShReadForceFb[i].Valid;
		gShuttleIf[i].Status.ShuttleInfo.Position.Value := Fbs.ShReadPositionFb[i].PositionInfo;
		gShuttleIf[i].Status.ShuttleInfo.Position.Valid := Fbs.ShReadPositionFb[i].Valid;
		gShuttleIf[i].Status.ShuttleInfo.State.Value := Fbs.ShReadState[i].State;
		gShuttleIf[i].Status.ShuttleInfo.State.Valid := Fbs.ShReadState[i].Valid;
	END_FOR;

	IF gAcp6DCtrlIf.Cmd.GetErrorInfo THEN
		Fbs.GetErrorCodesFb.Controller := ADR(gMcAcp6DController);
		Fbs.GetErrorCodesFb.Execute := TRUE;

		IF Fbs.GetErrorCodesFb.Valid OR Fbs.GetErrorCodesFb.Error THEN
			gAcp6DCtrlIf.Status.ErrorCodes := Fbs.GetErrorCodesFb.ErrorCodes;
			Fbs.GetErrorCodesFb.Execute := FALSE;
			gAcp6DCtrlIf.Cmd.GetErrorInfo := FALSE;
		END_IF

	END_IF

	Fbs.GetErrorCodesFb();
	Fbs.SysReadStateFb();
	Fbs.PowerOffFb();
	Fbs.PowerOnFb();
	Fbs.AutoRefreshFB();

	gAcp6DCtrlIf.Status.Ready := state = ACP6D_READY;
	gAcp6DCtrlIf.Status.Error := state = ACP6D_ERROR;
	gAcp6DCtrlIf.Status.ReadyToPowerOn := Fbs.SysReadStateFb.Valid AND Fbs.SysReadStateFb.State = mcACP6D_STATE_INACTIVE;

END_PROGRAM
```

#### Init.st
```iecst
PROGRAM _INIT
	gMcAcp6DController.H2P_START := ADR(FBout);
	gMcAcp6DController.P2H_START := ADR(FBin);
	gMcAcp6DController.ConfiguredFeedbackStreamAxis	:= 63;

	Fbs.AutoRefreshFB.Controller	:= ADR(gMcAcp6DController);
	Fbs.PowerOffFb.Controller := ADR(gMcAcp6DController);
	Fbs.PowerOnFb.Controller := ADR(gMcAcp6DController);
	Fbs.SysReadStateFb.Controller := ADR(gMcAcp6DController);

	Fbs.AutoRefreshFB.Enable := TRUE;
	Fbs.SysReadStateFb.Enable := TRUE;
END_PROGRAM
```

### Program Logical/Source/6DCtrl/MacroLoad (IEC)

#### Types.typ
```iecst
TYPE
	MacroLoadFbsTyp : 	STRUCT  (*Fbs for the macro load functionality*)
		MacroLoadFb : MC_BR_MacroLoad_Acp6D; (*FB to load a macro from an XML file*)
		MacroClearFb : MC_BR_MacroClear_Acp6D; (*FB to clear a defined macro*)
	END_STRUCT;
	MacroLoadStateEnum :
		(
		MACLOAD_IDLE, (*Idle state for the macro load process*)
		MACLOAD_LOAD, (*Load state for the macro load process*)
		MACLOAD_COUNT_CHECK, (*State to determine if we have finished the load of all macros*)
		MACLOAD_CLEAR, (*State to exectue a macro clear FB*)
		MACLOAD_DONE, (*State to denote completion of the initalize load process*)
		MACLOAD_ERROR (*Macro Load error state*)
		);
END_TYPE
```

#### Variables.var
```iecst
VAR
	state : MacroLoadStateEnum; (*state of the Macro Load process*)
	MacroFbs : MacroLoadFbsTyp; (*Function blocks for the macro load process*)
END_VAR
```

#### Cyclic.st
```iecst
PROGRAM _CYCLIC
	CASE state OF
		MACLOAD_IDLE:	//******************************************************************************** Macro Idle State
			IF gMacroLoadIf.Cmd.LoadAll OR gMacroLoadIf.Cmd.LoadSingle THEN
				gMacroLoadIf.Status.AllMacrosLoaded := FALSE;
				gMacroLoadIf.Status.Loading := TRUE;
				gMacroLoadIf.Status.CurrentMacro := 0;

				state := MACLOAD_COUNT_CHECK;
			ELSIF gMacroLoadIf.Cmd.Clear THEN
				MacroFbs.MacroClearFb.Controller := ADR(gMcAcp6DController);
				MacroFbs.MacroClearFb.MacroID := gMacroLoadIf.Par.SingleMacroLoad.MacroID;
				MacroFbs.MacroClearFb.Execute := TRUE;

				state := MACLOAD_CLEAR;
			ELSIF gMacroLoadIf.Cmd.Reset THEN
				gMacroLoadIf.Status.AllMacrosLoaded := FALSE;
				gMacroLoadIf.Cmd.Reset := FALSE;
			END_IF

		MACLOAD_LOAD://******************************************************************************** Macro Load State
			IF MacroFbs.MacroLoadFb.Error THEN
				gMacroLoadIf.Status.Error := TRUE;
				gMacroLoadIf.Status.MacroIDError := gMacroLoadIf.Status.CurrentMacro;

				state := MACLOAD_ERROR;
			ELSIF MacroFbs.MacroLoadFb.Done THEN
				MacroFbs.MacroLoadFb.Execute := FALSE;
				IF gMacroLoadIf.Cmd.LoadSingle THEN
					gMacroLoadIf.Status.CmdDone := TRUE;
				ELSE //Means we commanded a "LOAD ALL"
					gMacroLoadIf.Status.CurrentMacro := gMacroLoadIf.Status.CurrentMacro + 1;

					state := MACLOAD_COUNT_CHECK;
				END_IF
			END_IF

		MACLOAD_COUNT_CHECK: //******************************************************************************** Macro Count check State
			IF gMacroLoadIf.Par.MacroList[gMacroLoadIf.Status.CurrentMacro].Load THEN
				MacroFbs.MacroLoadFb.Controller := ADR(gMcAcp6DController);
				MacroFbs.MacroLoadFb.FileDevice := gMacroLoadIf.Par.FileDevice;
				IF gMacroLoadIf.Cmd.LoadAll THEN
					MacroFbs.MacroLoadFb.MacroID := gMacroLoadIf.Par.MacroList[gMacroLoadIf.Status.CurrentMacro].MacroID;
					MacroFbs.MacroLoadFb.FileName := gMacroLoadIf.Par.MacroList[gMacroLoadIf.Status.CurrentMacro].MacroFileName;

				ELSIF gMacroLoadIf.Cmd.LoadSingle THEN
					MacroFbs.MacroLoadFb.MacroID := gMacroLoadIf.Par.SingleMacroLoad.MacroID;
					MacroFbs.MacroLoadFb.FileName := gMacroLoadIf.Par.SingleMacroLoad.MacroFileName;
				END_IF
				MacroFbs.MacroLoadFb.Execute := TRUE;
				state := MACLOAD_LOAD;
			ELSE
				gMacroLoadIf.Status.CurrentMacro := gMacroLoadIf.Status.CurrentMacro + 1;
				IF gMacroLoadIf.Status.CurrentMacro >= MAX_MACRO_COUNT THEN
					gMacroLoadIf.Status.AllMacrosLoaded := TRUE;
					gMacroLoadIf.Status.CmdDone := TRUE;

					state := MACLOAD_DONE;
				END_IF
			END_IF
		MACLOAD_CLEAR: //******************************************************************************** Macro Clear state
			IF MacroFbs.MacroClearFb.Error THEN
				gMacroLoadIf.Status.Error := TRUE;

				state := MACLOAD_ERROR;
			ELSIF MacroFbs.MacroClearFb.Done THEN
				MacroFbs.MacroClearFb.Execute := FALSE;
				gMacroLoadIf.Status.CmdDone := TRUE;

				state := MACLOAD_DONE;
			END_IF
		MACLOAD_DONE: //******************************************************************************** Load Done State
			gMacroLoadIf.Status.Loading := FALSE;
			IF NOT gMacroLoadIf.Cmd.Clear AND NOT gMacroLoadIf.Cmd.LoadAll AND NOT gMacroLoadIf.Cmd.LoadSingle THEN
				gMacroLoadIf.Status.CmdDone := FALSE;
				state := MACLOAD_IDLE;
			END_IF
		MACLOAD_ERROR: //******************************************************************************** Macro load error State
			IF gMacroLoadIf.Cmd.Reset THEN
				MacroFbs.MacroClearFb.Execute := FALSE;
				MacroFbs.MacroLoadFb.Execute := FALSE;

				gMacroLoadIf.Cmd.Reset := FALSE;

				gMacroLoadIf.Status.Loading := FALSE;
				gMacroLoadIf.Status.AllMacrosLoaded := FALSE;
				gMacroLoadIf.Status.Error := FALSE;
				gMacroLoadIf.Status.MacroIDError := 0;
				state := MACLOAD_IDLE;
			END_IF
	END_CASE;

	//FB Calls
	MacroFbs.MacroLoadFb();
	MacroFbs.MacroClearFb();
END_PROGRAM
```

#### Init.st
```iecst
PROGRAM _INIT
	//Enable the macros for loading
	gMacroLoadIf.Par.MacroList[0].Load := TRUE;
	gMacroLoadIf.Par.MacroList[0].MacroFileName := '128_LoadToPrint.xml';
	gMacroLoadIf.Par.MacroList[0].MacroID := 128;

	gMacroLoadIf.Par.MacroList[1].Load := TRUE;
	gMacroLoadIf.Par.MacroList[1].MacroFileName := '129_PrintToDose1.xml';
	gMacroLoadIf.Par.MacroList[1].MacroID := 129;

	gMacroLoadIf.Par.MacroList[2].Load := TRUE;
	gMacroLoadIf.Par.MacroList[2].MacroFileName := '130_PrintToDose2.xml';
	gMacroLoadIf.Par.MacroList[2].MacroID := 130;

	gMacroLoadIf.Par.MacroList[3].Load := TRUE;
	gMacroLoadIf.Par.MacroList[3].MacroFileName := '131_DoseToPrint.xml';
	gMacroLoadIf.Par.MacroList[3].MacroID := 131;

	gMacroLoadIf.Par.MacroList[4].Load := TRUE;
	gMacroLoadIf.Par.MacroList[4].MacroFileName := '132_PrintToTamp.xml';
	gMacroLoadIf.Par.MacroList[4].MacroID := 132;

	gMacroLoadIf.Par.MacroList[5].Load := TRUE;
	gMacroLoadIf.Par.MacroList[5].MacroFileName := '133_TampToUnload.xml';
	gMacroLoadIf.Par.MacroList[5].MacroID := 133;

	gMacroLoadIf.Par.MacroList[6].Load := TRUE;
	gMacroLoadIf.Par.MacroList[6].MacroFileName := '134_UnloadToLoad.xml';
	gMacroLoadIf.Par.MacroList[6].MacroID := 134;

	gMacroLoadIf.Par.MacroList[7].Load := TRUE;
	gMacroLoadIf.Par.MacroList[7].MacroFileName := '135_RecoveryGroup0.xml';
	gMacroLoadIf.Par.MacroList[7].MacroID := 135;

	gMacroLoadIf.Par.MacroList[8].Load := TRUE;
	gMacroLoadIf.Par.MacroList[8].MacroFileName := '136_RecoveryGroup1.xml';
	gMacroLoadIf.Par.MacroList[8].MacroID := 136;

	gMacroLoadIf.Par.MacroList[9].Load := TRUE;
	gMacroLoadIf.Par.MacroList[9].MacroFileName := '137_RecoveryGroup2.xml';
	gMacroLoadIf.Par.MacroList[9].MacroID := 137;
	//Define the parameters for the macro load IF
	gMacroLoadIf.Par.FileDevice := '6DMacro';
END_PROGRAM
```

### Program Logical/Source/Auxil/AuditCtrl (IEC)

#### Variables.var
```iecst
VAR
	AuditCoreFb : MpAuditTrail;
END_VAR
```

#### Cyclic.st
```iecst
PROGRAM _CYCLIC
	AuditCoreFb.MpLink := ADR(gAuditTrail);
	AuditCoreFb.Enable := TRUE;
	AuditCoreFb.DeviceName := ADR('AuditFileDev');
	AuditCoreFb();

END_PROGRAM
```

### Program Logical/Source/Auxil/Vis (IEC)

#### Types.typ
```iecst
TYPE
	ShVisTyp : 	STRUCT
		ID : USINT;
		Visible : BOOL;
		Color : INT;
		Pos : McAcp6DShPositionInfoType;
		ScnViewer : ScnViewerConnectionTyp;
	END_STRUCT;
	VisTyp : {REDUND_UNREPLICABLE} 	STRUCT
		Shuttles : {REDUND_UNREPLICABLE} ARRAY[0..MAX_SHUTTLE_COUNT_ARRAY]OF ShVisTyp;
	END_STRUCT;
	VisShuttleStateEnum :
		(
		VIS_INIT,
		VIS_ACTIVE,
		VIS_ERROR
		);
	ScnViewerConnectionTyp : 	STRUCT
		EnablePositioner : USINT;
		EnablePath : BOOL;
		ClearPath : BOOL;
		PathColor : ScnViewerPathTyp;
	END_STRUCT;
	ScnViewerPathTyp : 	STRUCT
		Red : USINT;
		Green : USINT;
		Blue : USINT;
	END_STRUCT;
	ShuttleColorEnum :
		(
		COLOR_RED := 1,
		COLOR_BLUE_MATTE,
		COLOR_GREY_MATTE,
		COLOR_YELLOW_MATTE,
		COLOR_GREEN_MATTE,
		COLOR_ORANGE_MATTE,
		COLOR_WHITE_MATTE,
		COLOR_BLACK_MATTE
		);
END_TYPE
```

#### Variables.var
```iecst
VAR
	Vis : VisTyp;
	ShData : ARRAY[0..9] OF MC_BR_ShReadPosition_Acp6D;
	states : ARRAY[0..9] OF VisShuttleStateEnum;
	idx : USINT;
END_VAR
```

#### Cyclic.st
```iecst
PROGRAM _CYCLIC
	FOR idx := 0 TO gMainIf.Cfg.ShuttleCount - 1 DO
		IF Vis.Shuttles[idx].ID <> 0 THEN
			Vis.Shuttles[idx].Visible := TRUE;
			Vis.Shuttles[idx].Pos.X := gShuttleIf[idx].Status.ShuttleInfo.Position.Value.X * 1000;
			Vis.Shuttles[idx].Pos.Y := gShuttleIf[idx].Status.ShuttleInfo.Position.Value.Y * 1000;
			Vis.Shuttles[idx].Pos.Z := gShuttleIf[idx].Status.ShuttleInfo.Position.Value.Z * 1000;
			Vis.Shuttles[idx].Pos.RX := gShuttleIf[idx].Status.ShuttleInfo.Position.Value.RX / 3.14189 * 180.0;
			Vis.Shuttles[idx].Pos.RY := gShuttleIf[idx].Status.ShuttleInfo.Position.Value.RY / 3.14189 * 180.0;
			Vis.Shuttles[idx].Pos.RZ := gShuttleIf[idx].Status.ShuttleInfo.Position.Value.RZ / 3.14189 * 180.0;
			CASE gShuttleIf[idx].Status.ShuttleInfo.State.Value OF
				mcACP6D_SH_STATE_UNDETECTED: (*Shuttle is not detected by the System*)
					Vis.Shuttles[idx].Color := DINT_TO_INT(COLOR_GREY_MATTE);
				mcACP6D_SH_STATE_DISCOVERING: (*Shuttle iis in the process of being discovered by the System		*)
				mcACP6D_SH_STATE_LANDED :  (*Shuttle is landed and controlled by the System. 			*)
					Vis.Shuttles[idx].Color := DINT_TO_INT(COLOR_BLUE_MATTE);
				mcACP6D_SH_STATE_IDLING :  (*Shuttle is levitating and not currently executing a motion command		*)
					Vis.Shuttles[idx].Color := DINT_TO_INT(COLOR_WHITE_MATTE);
				mcACP6D_SH_STATE_DISABLED :  (*Shuttle is not controlled by the System		*)
				mcACP6D_SH_STATE_MOTION :  (*Shuttle is in motion		*)
					Vis.Shuttles[idx].Color := DINT_TO_INT(COLOR_WHITE_MATTE);
				mcACP6D_SH_STATE_WAIT :  (*Shuttle is waiting for a trigger defined by the WaitUntil command		*)
				mcACP6D_SH_STATE_STOPPING :  (*Shuttle is performing an automatic quick stop due to obstacle detection		*)
				mcACP6D_SH_STATE_OBSTACLE :  (*Shuttle is waiting for an obstacle to clear before proceeding*)
					Vis.Shuttles[idx].Color := DINT_TO_INT(COLOR_YELLOW_MATTE);
				mcACP6D_SH_STATE_HOLD :  (*Shuttle is holding position due to positioning error		*)
				mcACP6D_SH_STATE_STOPPED :  (*Shuttle is stopped due to obstacle or boundary detection, it  cannot automatically resume its motion		*)
				mcACP6D_SH_STATE_ERROR :  (*Shuttle has detected an error		*)
					Vis.Shuttles[idx].Color := DINT_TO_INT(COLOR_RED);
				mcACP6D_SH_STATE_RESERVED :  (*Reserved State*)
			END_CASE;
		ELSE
			Vis.Shuttles[idx].Visible := TRUE;
		END_IF
	END_FOR;
END_PROGRAM
```

#### Init.st
```iecst
PROGRAM _INIT
	FOR idx := 0 TO gMainIf.Cfg.ShuttleCount - 1 DO
		Vis.Shuttles[idx].ID := idx+1;
	END_FOR;
END_PROGRAM
```

### Program Logical/Source/Auxil/OeeCalc (IEC)

#### Cyclic.st - Cyclic code
```iecst
PROGRAM _CYCLIC

	SysThroughputCalcFb.Enable := gProcessInfoIf.Cmd.Enable;
	SysThroughputCalcFb.ProductCounter := gProcessInfoIf.Par.CurrentProductCount;
	SysThroughputCalcFb.Reset := gProcessInfoIf.Cmd.ResetData;

	PowThroughputCalcFb.Enable := gProcessInfoIf.Cmd.Enable;
	PowThroughputCalcFb.ProductCounter := gProcessInfoIf.Par.CurrentPowderCount;
	PowThroughputCalcFb.Reset := gProcessInfoIf.Cmd.ResetData;

	gProcessInfoIf.Sts.Enabled := gProcessInfoIf.Cmd.Enable;
	IF gProcessInfoIf.Cmd.ResetData THEN
		gProcessInfoIf.Cmd.ResetData := FALSE;
		gProcessInfoIf.Par.CurrentProductCount := 0;
	END_IF

	SysThroughputCalcFb();
	PowThroughputCalcFb();

	gProcessInfoIf.Sts.CurrentBlistersPerMinute := SysThroughputCalcFb.PPM * 6;
	//gProcessInfoIf.Sts.CurrentLayersPerMinute := SysThroughputCalcFb.PPM * 4;
	gProcessInfoIf.Sts.CurrentLayersPerMinute := PowThroughputCalcFb.PPM / 3;

	gProcessInfoIf.Sts.CurrentPPM := SysThroughputCalcFb.PPM;
	gProcessInfoIf.Sts.CurrentPPH := SysThroughputCalcFb.PPH;

END_PROGRAM
```

#### Types.typ - Local data types
```iecst
TYPE
	ProcThroughputTyp : 	STRUCT
		Enable : BOOL;
		Reset : BOOL;
		ProductCounter : UDINT;
		New_Member : USINT;
	END_STRUCT;
	ThroughputCalcInternalTyp : 	STRUCT
		startTime : UDINT;
		state : ThroughputCalcInternalStateEnum;
		timeSinceStart : TIME;
		AvgCycleTimeUdint : UDINT;
	END_STRUCT;
	ThroughputCalcInternalStateEnum :
		(
		TC_OFF,
		TC_INIT,
		TC_CALC,
		TC_ERROR
		);
END_TYPE
```

#### Variables.var - Local variables
```iecst
VAR
	SysThroughputCalcFb : ThroughputCounterFb;
	PowThroughputCalcFb : ThroughputCounterFb;
END_VAR
```

#### LocalFunctions.fun
```iecst
{REDUND_ERROR} FUNCTION_BLOCK ThroughputCounterFb (*Function block that provides a simple PPM calculator*) (*$GROUP=User,$CAT=User,$GROUPICON=User.png,$CATICON=User.png*)
	VAR_INPUT
		Enable : BOOL; (*Enable the calculation*)
		Reset : BOOL; (*Reset the buffer values*)
		ProductCounter : UDINT; (*Product counter*)
	END_VAR
	VAR_OUTPUT
		AvgCycleTime : {REDUND_UNREPLICABLE} TIME; (*Calculated avergage cycle time per product*)
		PPM : {REDUND_UNREPLICABLE} REAL; (*Extrapolated calculation of PPM*)
		PPH : {REDUND_UNREPLICABLE} REAL; (*Extrapolated calculation of PPH*)
	END_VAR
	VAR
		Internal : {REDUND_UNREPLICABLE} ThroughputCalcInternalTyp;
	END_VAR
END_FUNCTION_BLOCK
```

#### ThroughputCounterFb.st
```iecst
(* TODO: Add your comment here *)
FUNCTION_BLOCK ThroughputCounterFb
	CASE Internal.state OF
		TC_OFF:
			IF Enable THEN
				Internal.state := TC_INIT;
			END_IF
		TC_INIT:
			Internal.startTime := TIME_TO_UDINT(clock_ms());	//Determine start clock
			Internal.state := TC_CALC;
		TC_CALC:
			IF Reset THEN 	//Head back to the init state and reset internal start time
				Reset := FALSE;
				Internal.state := TC_INIT;
			ELSIF NOT Enable THEN	//Disable if the enable is dropped
				AvgCycleTime := 0;
				Internal.AvgCycleTimeUdint := 0;
				Internal.timeSinceStart := 0;
				Internal.state := TC_OFF;
			ELSIF ProductCounter <> 0 THEN //Done to ensure no divide by 0
				Internal.timeSinceStart := (TIME_TO_UDINT(clock_ms()) - Internal.startTime);	//Calculate time since the start of the monitoring
				AvgCycleTime := Internal.timeSinceStart / ProductCounter;	//Calculate current estimated cycle time
				Internal.AvgCycleTimeUdint := TIME_TO_UDINT(AvgCycleTime);	//Convert to a UDINT
				PPM := 60.0 * 1 / (Internal.AvgCycleTimeUdint / 1000.0);	//Calculate PPM
				PPH := 3600.0 * 1 / (Internal.AvgCycleTimeUdint / 1000.0);	//Calculate PPH
			END_IF
		TC_ERROR:
			IF NOT Enable THEN
				AvgCycleTime := 0;
				Internal.AvgCycleTimeUdint := 0;
				Internal.timeSinceStart := 0;
				Internal.state := TC_OFF;
			END_IF
	END_CASE;
END_FUNCTION_BLOCK
```

### Program Logical/Source/Auxil/SVControl

#### Types.typ
```iecst
TYPE
	MoveType_enum :
		(
		LINEAR,
		RADIAL
		);
	Binding_typ : 	STRUCT
		Camera : SceneViewCamera_typ;
		FocalPoint : SceneViewCoord_typ;
		FocalPointVisible : BOOL;
	END_STRUCT;
	Vis_typ : 	STRUCT
		Controls : Controls_typ;
		Bind : Binding_typ;
	END_STRUCT;
	LinearControls_typ : 	STRUCT
		XBtnPos : USINT;
		XBtnNeg : USINT;
		YBtnPos : USINT;
		YBtnNeg : USINT;
		Y : REAL;
		X : REAL;
	END_STRUCT;
	CircularControls_typ : 	STRUCT
		RadiusBtnNeg : USINT;
		RadiusBtnPos : USINT;
		Angle : REAL;
		Radius : REAL;
	END_STRUCT;
	Controls_typ : 	STRUCT
		FocalPoint : FocalPointControls_typ;
		Fov : REAL;
		Z : REAL;
		Circular : CircularControls_typ;
		Linear : LinearControls_typ;
		SavePointA : BOOL;
		MoveType : USINT;
		NewMove : BOOL;
		Start : BOOL;
		Load : BOOL;
		Save : BOOL;
		SelectedMove : USINT;
		MoveMode : MoveType_enum;
		TimeInput : REAL;
		ActiveMoveTravelTime : TIME;
		ActiveMoveElapsedTime : TIME;
		Pause : BOOL;
	END_STRUCT;
	FocalPointControls_typ : 	STRUCT
		XBtnPos : USINT;
		XBtnNeg : USINT;
		YBtnPos : USINT;
		YBtnNeg : USINT;
		ZBtnPos : USINT;
		ZBtnNeg : USINT;
		Visible : BOOL;
	END_STRUCT;
	Move_typ : 	STRUCT
		IsSaved : BOOL;
		MoveType : MoveType_enum;
		Point : SceneViewCamera_typ;
		FocalPoint : SceneViewCoord_typ;
		TravelTime : TIME;
	END_STRUCT;
	State_enum :
		(
		MOVE_SETTINGS,
		NEW_MOVE,
		UPDATE_LIST,
		REBUILD_LIST,
		NEW_MOVE_SAVE,
		SAVE_MOVE,
		LOAD_MOVE,
		START_MOVE,
		LINEAR_MOVE,
		WAIT_FOR_LINEAR_MOVE_DONE,
		RADIAL_MOVE,
		WAIT_FOR_RADIAL_MOVE_DONE,
		MOVE_COMPLETE,
		SAVE_LOAD_RECIPE,
		WAIT_FOR_STOP
		);
	RecipeCtrlTyp : 	STRUCT
		Cmd : RecipeCtrlCmdTyp;
		Par : RecipeCtrlParTyp;
		Sts : RecipeCtrlStsTyp;
	END_STRUCT;
	RecipeCtrlCmdTyp : 	STRUCT
		Save : BOOL;
		Load : BOOL;
	END_STRUCT;
	RecipeCtrlParTyp : 	STRUCT
		FileName : STRING[80];
	END_STRUCT;
	RecipeCtrlStsTyp : 	STRUCT
		LastLoadedRecipe : STRING[80];
	END_STRUCT;
END_TYPE
```

#### Variables.var
```iecst
VAR
	MoveText : STRING[80];
	RadialMove : SV_BE_RadialMove;
	FocalPointMove : SV_BE_FocalPointMove;
	State : State_enum;
	TravelTime : TIME := T#5s;
	Vis : Vis_typ := (Controls:=(TimeInput:=5),Bind:=(FocalPointVisible:=TRUE));
	FocalPointInit : SceneViewCoord_typ := (X:=1146,Y:=-743,Z:=-4);
	StartView : SceneViewCamera_typ := (Perspective:=TRUE,Zoom:=10,Fov:=61.9,ViewPoint:=(X:=-96,Y:=727,Z:=1140),ViewVector:=(X:=1.242,Y:=-1.47,Z:=-1.144),OrientationVector:=(X:=0,Y:=0,Z:=1));
	AngleRad : REAL;
	PointA : SceneViewCamera_typ;
	PointB : SceneViewCamera_typ;
	TotalNumMoves : USINT;
	CompletedMoves : USINT;
	Point : ARRAY[0..2] OF SceneViewCamera_typ;
END_VAR
VAR CONSTANT
	MAX_NUM_MOVES : USINT := 50;
END_VAR
VAR
	MoveNumText : ARRAY[0..MAX_NUM_MOVES] OF STRING[80];
	MoveIndexString : STRING[80];
	IntermediateDateProvider : ARRAY[0..MAX_NUM_MOVES] OF STRING[80];
	DataProvider : ARRAY[0..MAX_NUM_MOVES] OF STRING[80];
	CamMove : ARRAY[0..MAX_NUM_MOVES] OF Move_typ;
	i : USINT;
	FocalPointB : SceneViewCoord_typ;
	FocalPointA : SceneViewCoord_typ;
	SvMovieRecipeFb : MpRecipeXml;
	SvMovieRecipeRegParFb : MpRecipeRegPar;
	svMovieRecipeIf : RecipeCtrlTyp;
END_VAR
```

#### Main.st
```iecst
PROGRAM _INIT
	(* Insert code here *)

	Point[0] := StartView;
	Vis.Bind.Camera := StartView;

	Vis.Bind.FocalPoint.X := FocalPointInit.X;
	Vis.Bind.FocalPoint.Y := FocalPointInit.Y;
	Vis.Bind.FocalPoint.Z := FocalPointInit.Z;

	Vis.Controls.Linear.X := StartView.ViewPoint.X;
	Vis.Controls.Linear.Y := StartView.ViewPoint.Y;
	Vis.Controls.Z := StartView.ViewPoint.Z;
	Vis.Controls.Fov := StartView.Fov;
	Vis.Controls.Circular.Radius := 100;

	SvMovieRecipeFb.MpLink := ADR(gRecipeScnViewer);
	SvMovieRecipeFb.Enable := TRUE;
	SvMovieRecipeFb.Category := ADR('SvMovie');
	SvMovieRecipeFb.DeviceName := ADR('SvMovie');
	SvMovieRecipeFb.FileName := ADR(svMovieRecipeIf.Par.FileName);
	SvMovieRecipeFb();

	SvMovieRecipeRegParFb.MpLink := ADR(gRecipeScnViewer);
	SvMovieRecipeRegParFb.Enable := TRUE;
	SvMovieRecipeRegParFb.Category := ADR('SvMovie');
	SvMovieRecipeRegParFb.PVName := ADR('SVControl:CamMove');
	SvMovieRecipeRegParFb();
END_PROGRAM

PROGRAM _CYCLIC
	Vis.Bind.FocalPoint.X := Vis.Bind.FocalPoint.X + Vis.Controls.FocalPoint.XBtnPos - Vis.Controls.FocalPoint.XBtnNeg;
	Vis.Bind.FocalPoint.Y := Vis.Bind.FocalPoint.Y + Vis.Controls.FocalPoint.YBtnPos - Vis.Controls.FocalPoint.YBtnNeg;
	Vis.Bind.FocalPoint.Z := Vis.Bind.FocalPoint.Z + Vis.Controls.FocalPoint.ZBtnPos - Vis.Controls.FocalPoint.ZBtnNeg;

	Vis.Controls.Circular.Radius := Vis.Controls.Circular.Radius + Vis.Controls.Circular.RadiusBtnPos - Vis.Controls.Circular.RadiusBtnNeg;
	Vis.Controls.Linear.X := Vis.Controls.Linear.X + Vis.Controls.Linear.XBtnPos - Vis.Controls.Linear.XBtnNeg;
	Vis.Controls.Linear.Y := Vis.Controls.Linear.Y + Vis.Controls.Linear.YBtnPos - Vis.Controls.Linear.YBtnNeg;

	Vis.Bind.FocalPointVisible := Vis.Controls.FocalPoint.Visible;

	CASE State OF
		MOVE_SETTINGS: //set points
			CASE Vis.Controls.MoveMode OF
				LINEAR:
					MoveText := 'Linear';
					Vis.Bind.Camera.ViewPoint.X := Vis.Controls.Linear.X;
					Vis.Bind.Camera.ViewPoint.Y := Vis.Controls.Linear.Y;

					//keeps view the same when switching to radial mode
					AngleRad := atan2((Vis.Bind.Camera.ViewPoint.Y - Vis.Bind.FocalPoint.Y),(Vis.Bind.Camera.ViewPoint.X - Vis.Bind.FocalPoint.X));
					Vis.Controls.Circular.Angle := AngleRad * 180 / PI;
					IF Vis.Controls.Circular.Angle < 0 THEN
						Vis.Controls.Circular.Angle := Vis.Controls.Circular.Angle + 360;
					ELSIF Vis.Controls.Circular.Angle >= 360 THEN
						Vis.Controls.Circular.Angle := Vis.Controls.Circular.Angle - 360;
					END_IF
					Vis.Controls.Circular.Radius := (Vis.Bind.Camera.ViewPoint.X - Vis.Bind.FocalPoint.X) / COS(AngleRad);
				RADIAL:
					MoveText := 'Radial';
					AngleRad := Vis.Controls.Circular.Angle * PI / 180;

					Vis.Bind.Camera.ViewPoint.X := (Vis.Controls.Circular.Radius * COS(AngleRad)) + Vis.Bind.FocalPoint.X;
					Vis.Bind.Camera.ViewPoint.Y := (Vis.Controls.Circular.Radius * SIN(AngleRad)) + Vis.Bind.FocalPoint.Y;

					Vis.Controls.Linear.X := Vis.Bind.Camera.ViewPoint.X;
					Vis.Controls.Linear.Y := Vis.Bind.Camera.ViewPoint.Y;
			END_CASE

			Vis.Bind.Camera.OrientationVector.X := 0;
			Vis.Bind.Camera.OrientationVector.Y := 0;
			Vis.Bind.Camera.OrientationVector.Z := 1;

			Vis.Bind.Camera.ViewPoint.Z := Vis.Controls.Z;
			Vis.Bind.Camera.Fov := Vis.Controls.Fov;

			Vis.Bind.Camera.ViewVector.X := (Vis.Bind.FocalPoint.X - Vis.Bind.Camera.ViewPoint.X) / 1000.0;
			Vis.Bind.Camera.ViewVector.Y := (Vis.Bind.FocalPoint.Y - Vis.Bind.Camera.ViewPoint.Y) / 1000.0;
			Vis.Bind.Camera.ViewVector.Z := (Vis.Bind.FocalPoint.Z - Vis.Bind.Camera.ViewPoint.Z) / 1000.0;

			IF Vis.Controls.NewMove THEN
				Vis.Controls.NewMove := FALSE;
				State := NEW_MOVE;
			ELSIF Vis.Controls.Load THEN
				State := LOAD_MOVE;
			ELSIF Vis.Controls.Save THEN
				Vis.Controls.Save := FALSE;
				State := SAVE_MOVE;
			END_IF

			IF svMovieRecipeIf.Cmd.Load OR svMovieRecipeIf.Cmd.Save THEN
				SvMovieRecipeFb.Save := svMovieRecipeIf.Cmd.Save;
				SvMovieRecipeFb.Load := svMovieRecipeIf.Cmd.Load;

				State := SAVE_LOAD_RECIPE;
			END_IF

			IF Vis.Controls.SavePointA THEN
				Vis.Controls.SavePointA := FALSE;
				Point[0] := Vis.Bind.Camera;
			END_IF

			IF Vis.Controls.Start THEN
				CompletedMoves := 0;
				PointA := Point[0];
				PointB := CamMove[0].Point;
				FocalPointA := FocalPointInit;
				FocalPointB := CamMove[0].FocalPoint;
				State := START_MOVE;
			END_IF

		NEW_MOVE: //new move
			FOR i := 0 TO MAX_NUM_MOVES DO
				IF NOT CamMove[i].IsSaved THEN
					CamMove[i].IsSaved := TRUE;
					CamMove[i].MoveType := Vis.Controls.MoveMode;
					CamMove[i].TravelTime := REAL_TO_TIME(Vis.Controls.TimeInput * 1000);

					State := NEW_MOVE_SAVE;
					EXIT;
				ELSIF i = MAX_NUM_MOVES THEN
					State := MOVE_SETTINGS;
				END_IF
			END_FOR

		NEW_MOVE_SAVE:

			TotalNumMoves := TotalNumMoves + 1;
			CamMove[i].Point := Vis.Bind.Camera;
			CamMove[i].FocalPoint := Vis.Bind.FocalPoint;

			State := UPDATE_LIST;

		UPDATE_LIST:
			brsftoa(i, ADR(MoveIndexString));
			MoveNumText[i] := CONCAT(MoveIndexString, ': ');
			MoveNumText[i] := CONCAT(MoveNumText[i], MoveText);
			MoveNumText[i] := CONCAT(MoveNumText[i], ' Move');

			IntermediateDateProvider[i] := CONCAT('{"value":"',MoveIndexString);
			IntermediateDateProvider[i] := CONCAT(IntermediateDateProvider[i],'","text":"');
			IntermediateDateProvider[i] := CONCAT(IntermediateDateProvider[i], MoveNumText[i]);
			DataProvider[i] := CONCAT(IntermediateDateProvider[i],'"}');

			State := MOVE_SETTINGS;
		SAVE_LOAD_RECIPE:
			IF SvMovieRecipeFb.CommandDone THEN
				IF svMovieRecipeIf.Cmd.Load THEN
					SvMovieRecipeFb.Load := FALSE;
					svMovieRecipeIf.Cmd.Load := FALSE;
					svMovieRecipeIf.Sts.LastLoadedRecipe := svMovieRecipeIf.Par.FileName;

					State := REBUILD_LIST;
				ELSIF svMovieRecipeIf.Cmd.Save THEN
					SvMovieRecipeFb.Save := FALSE;
					svMovieRecipeIf.Cmd.Save := FALSE;

					State := MOVE_SETTINGS;
				END_IF
			END_IF
		REBUILD_LIST:
			brsmemset(ADR(DataProvider),0,SIZEOF(DataProvider));
			brsmemset(ADR(MoveNumText),0,SIZEOF(MoveNumText));
			brsmemset(ADR(IntermediateDateProvider),0,SIZEOF(IntermediateDateProvider));
			TotalNumMoves := 0; //Added for loading saved recipes
			FOR i:=0 TO MAX_NUM_MOVES DO
				IF CamMove[i].IsSaved THEN
					TotalNumMoves := TotalNumMoves + 1;
					brsftoa(i, ADR(MoveIndexString));
					MoveNumText[i] := CONCAT(MoveIndexString, ': ');
					CASE CamMove[i].MoveType OF
						LINEAR:
							MoveNumText[i] := CONCAT(MoveNumText[i], 'Linear');
						RADIAL:
							MoveNumText[i] := CONCAT(MoveNumText[i], 'Radial');
					END_CASE;
					MoveNumText[i] := CONCAT(MoveNumText[i], ' Move');

					IntermediateDateProvider[i] := CONCAT('{"value":"',MoveIndexString);
					IntermediateDateProvider[i] := CONCAT(IntermediateDateProvider[i],'","text":"');
					IntermediateDateProvider[i] := CONCAT(IntermediateDateProvider[i], MoveNumText[i]);
					DataProvider[i] := CONCAT(IntermediateDateProvider[i],'"}');
				END_IF
			END_FOR;

			State := MOVE_SETTINGS;
		LOAD_MOVE: //load
			Vis.Controls.Load := FALSE;

			IF CamMove[Vis.Controls.SelectedMove].IsSaved THEN
				Vis.Controls.Linear.X := CamMove[Vis.Controls.SelectedMove].Point.ViewPoint.X;
				Vis.Controls.Linear.Y := CamMove[Vis.Controls.SelectedMove].Point.ViewPoint.Y;

				Vis.Controls.Z := CamMove[Vis.Controls.SelectedMove].Point.ViewPoint.Z;
				Vis.Controls.Fov := CamMove[Vis.Controls.SelectedMove].Point.Fov;
				Vis.Controls.TimeInput := TIME_TO_REAL(CamMove[Vis.Controls.SelectedMove].TravelTime) / 1000;
				Vis.Controls.MoveMode := CamMove[Vis.Controls.SelectedMove].MoveType;

				Vis.Bind.Camera := CamMove[Vis.Controls.SelectedMove].Point;
				Vis.Bind.FocalPoint := CamMove[Vis.Controls.SelectedMove].FocalPoint;

				//update radial controls
				AngleRad := atan2((Vis.Bind.Camera.ViewPoint.Y - Vis.Bind.FocalPoint.Y),(Vis.Bind.Camera.ViewPoint.X - Vis.Bind.FocalPoint.X));
				Vis.Controls.Circular.Angle := AngleRad * 180 / PI;
				IF Vis.Controls.Circular.Angle < 0 THEN
					Vis.Controls.Circular.Angle := Vis.Controls.Circular.Angle + 360;
				ELSIF Vis.Controls.Circular.Angle >= 360 THEN
					Vis.Controls.Circular.Angle := Vis.Controls.Circular.Angle - 360;
				END_IF
				Vis.Controls.Circular.Radius := (Vis.Bind.Camera.ViewPoint.X - Vis.Bind.FocalPoint.X) / COS(AngleRad);

			END_IF
			State := MOVE_SETTINGS;

		SAVE_MOVE: //save
			IF CamMove[Vis.Controls.SelectedMove].IsSaved THEN
				CamMove[Vis.Controls.SelectedMove].Point := Vis.Bind.Camera;
				CamMove[Vis.Controls.SelectedMove].FocalPoint := Vis.Bind.FocalPoint;
				CamMove[Vis.Controls.SelectedMove].TravelTime := REAL_TO_TIME(Vis.Controls.TimeInput * 1000);
				i := Vis.Controls.SelectedMove;
				State := UPDATE_LIST;
			ELSE
				State := MOVE_SETTINGS;
			END_IF

		START_MOVE:
			TravelTime := CamMove[CompletedMoves].TravelTime;
			IF CamMove[CompletedMoves].MoveType = LINEAR THEN
				State := LINEAR_MOVE;
			ELSIF CamMove[CompletedMoves].MoveType = RADIAL THEN
				State := RADIAL_MOVE;
			END_IF

		RADIAL_MOVE:
			Vis.Controls.SelectedMove := CompletedMoves;
			RadialMove.PointA := PointA;
			RadialMove.PointB := PointB;
			RadialMove.FocalPointA := FocalPointA;
			RadialMove.FocalPointB := FocalPointB;
			RadialMove.TravelTime := TravelTime;
			RadialMove.Execute := TRUE;
			State := WAIT_FOR_RADIAL_MOVE_DONE;

		WAIT_FOR_RADIAL_MOVE_DONE:
			IF RadialMove.Done AND NOT Vis.Controls.Pause THEN
				RadialMove.Execute := FALSE;
				CompletedMoves := CompletedMoves + 1;
				State := MOVE_COMPLETE;
			END_IF

			RadialMove();
			Vis.Controls.ActiveMoveTravelTime := TravelTime;
			Vis.Controls.ActiveMoveElapsedTime := RadialMove.ElapsedTime;
			Vis.Bind.FocalPoint := RadialMove.FocalPointPos;
			Vis.Bind.Camera := RadialMove.SceneViewPos;

		LINEAR_MOVE:
			Vis.Controls.SelectedMove := CompletedMoves;
			FocalPointMove.PointA := PointA;
			FocalPointMove.PointB := PointB;
			//FocalPointMove.FocalPoint := Vis.FocalPoint;
			FocalPointMove.FocalPointA := FocalPointA;
			FocalPointMove.FocalPointB := FocalPointB;
			FocalPointMove.TravelTime := TravelTime;
			FocalPointMove.Execute := TRUE;
			State := WAIT_FOR_LINEAR_MOVE_DONE;

		WAIT_FOR_LINEAR_MOVE_DONE:

			IF FocalPointMove.Done AND NOT Vis.Controls.Pause THEN
				FocalPointMove.Execute := FALSE;
				CompletedMoves := CompletedMoves + 1;
				State := MOVE_COMPLETE;
			END_IF

			FocalPointMove();
			Vis.Controls.ActiveMoveTravelTime := TravelTime;
			Vis.Controls.ActiveMoveElapsedTime := FocalPointMove.ElapsedTime;
			Vis.Bind.FocalPoint := FocalPointMove.FocalPointPos;
			Vis.Bind.Camera := FocalPointMove.SceneViewPos;

		MOVE_COMPLETE:
			IF CompletedMoves < TotalNumMoves THEN
				PointA := Vis.Bind.Camera;
				PointB := CamMove[CompletedMoves].Point;
				FocalPointA := Vis.Bind.FocalPoint;
				FocalPointB := CamMove[CompletedMoves].FocalPoint;
				State := START_MOVE;
			ELSE
				State := WAIT_FOR_STOP;
			END_IF

		WAIT_FOR_STOP:
			IF NOT Vis.Controls.Start THEN
				State := MOVE_SETTINGS;
			END_IF
	END_CASE

	SvMovieRecipeFb();
	SvMovieRecipeRegParFb();

END_PROGRAM

PROGRAM _EXIT
	(* Insert code here *)

END_PROGRAM
```

### Program Logical/Source/Robots/RobotCtrl (IEC)

#### Types.typ
```iecst
TYPE
	RobotStateEnum :
		(
		RBT_OFF,
		RBT_INIT,
		RBT_HOME,
		RBT_POWER,
		RBT_IDLE,
		RBT_RUN_PROGRAM,
		RBT_DONE,
		RBT_ERROR
		);
END_TYPE
```

#### Variables.var
```iecst
VAR
	setProduct : BOOL;
	resetProduct : BOOL;
	DeltaFb : MpDelta3Axis;
	DeltaPars : MpDelta3AxisParType;
	state : RobotStateEnum;
	pRobotIf : REFERENCE TO RbtIfTyp;
	taskName : STRING[10];
	i : INT;
END_VAR
```

#### Cyclic.st
```iecst
PROGRAM _CYCLIC
	DeltaFb.Override := 100;
	DeltaFb.Parameters := ADR(DeltaPars);

	CASE state OF
		RBT_OFF:
			IF pRobotIf.Cmd.Enable THEN
				state := RBT_INIT;
			END_IF
		RBT_INIT:
			DeltaFb.Home := TRUE;
			state := RBT_HOME;
		RBT_HOME:
			IF DeltaFb.IsHomed THEN
				DeltaFb.Home := FALSE;
				DeltaFb.Power := TRUE;
				state := RBT_POWER;
			END_IF
		RBT_POWER:
			IF DeltaFb.PowerOn THEN
				pRobotIf.Sts.Powered := TRUE;
				pRobotIf.Sts.Ready := TRUE;
				state := RBT_IDLE;
			END_IF
		RBT_IDLE:
			IF NOT pRobotIf.Cmd.Enable THEN
				DeltaFb.Power := FALSE;
				state := RBT_OFF;
			ELSIF pRobotIf.Cmd.Run THEN
				DeltaFb.MoveProgram := TRUE;
				pRobotIf.Sts.Running := TRUE;
				state := RBT_RUN_PROGRAM;
			END_IF
		RBT_RUN_PROGRAM:
			IF setProduct THEN
				setProduct := FALSE;
				FOR i:=0 TO 3 DO
					pRobotIf.Par.Products[i].Present := TRUE;
				END_FOR;
			END_IF
			IF resetProduct THEN
				resetProduct := FALSE;
				FOR i:=0 TO 3 DO
					pRobotIf.Par.Products[i].Present := FALSE;
				END_FOR;
			END_IF
			IF DeltaFb.MoveDone THEN
				DeltaFb.MoveProgram := FALSE;
				pRobotIf.Sts.Running := FALSE;
				pRobotIf.Sts.Done := TRUE;

				state := RBT_DONE;
			END_IF
		RBT_DONE:
			IF NOT pRobotIf.Cmd.Run THEN
				pRobotIf.Sts.Done := FALSE;
				state := RBT_IDLE;
			END_IF
		RBT_ERROR:
			IF pRobotIf.Cmd.Reset THEN
				DeltaFb.ErrorReset := TRUE;
				IF NOT DeltaFb.Error THEN
					DeltaFb.ErrorReset := FALSE;
					pRobotIf.Cmd.Reset := FALSE;
					state := RBT_OFF;
				END_IF
			END_IF
	END_CASE;
	DeltaFb();
END_PROGRAM
```

#### Exit.st
```iecst
PROGRAM _EXIT
	DeltaFb.Enable := FALSE;
	DeltaFb();

END_PROGRAM
```

#### Init.st
```iecst
PROGRAM _INIT
	ST_name(0,ADR(taskName),0);

	IF taskName = 'LoadRbt' THEN
		pRobotIf ACCESS ADR(gRobotIf[Load_Robot]);
		DeltaPars.ProgramName := 'LoadPick.st';
		DeltaFb.MpLink := ADR(g3AxDeltaLoad);
	ELSIF taskName = 'UnloadRbt' THEN
		pRobotIf ACCESS ADR(gRobotIf[Unload_Robot]);
		DeltaPars.ProgramName := 'UnloadPick.st';
		DeltaFb.MpLink := ADR(g3AxDeltaUnload);
	END_IF
	DeltaFb.Enable := TRUE;

END_PROGRAM
```

### LoadPick.st
```iecst
VAR CONSTANT
	Rest : McPointType := (Pos:=(X:=0, Y:=0, Z:=-790));
	PlaceApproach : McPointType := (Pos:=(X:=60, Y:=0, Z:=-800));
	Place : McPointType := (Pos:=(X:=60, Y:=0, Z:=-850));
	PickApproach : McPointType := (Pos:=(X:=-300, Y:=0, Z:=-800));
	Pick : McPointType := (Pos:=(X:=-300, Y:=0, Z:=-900));

END_VAR
VAR{AT 'LoadStatio'}
	setLoad : BOOL;
	release : BOOL;
END_VAR
VAR{AT 'LoadRbt'}
	setProduct : BOOL;
END_VAR
PROGRAM _MAIN
	Feedrate(100000);
	MoveL(Rest);
	RoundingEdges(50);
	MoveL(PlaceApproach);
	MoveLR(Place);
	DO_PATH_SYNCH
		setLoad := TRUE;
	END_PATH_SYNCH
	WaitTime(0.2);
	DO_PATH_SYNCH
		release := TRUE;
	END_PATH_SYNCH
	RoundingEdges(50);
	MoveL(PlaceApproach);
	MoveL(PickApproach);
	MoveL(Pick);
	WaitTime(0.2);
	DO_PATH_SYNCH
		setProduct := TRUE;
	END_PATH_SYNCH
	MoveL(PickApproach);
	MoveL(Rest);
END_PROGRAM
```

### UnloadPick.st
```iecst
VAR CONSTANT
	Rest : McPointType := (Pos:=(X:=0, Y:=0, Z:=-790));
	PlaceApproach : McPointType := (Pos:=(X:=300, Y:=0, Z:=-800));
	Place : McPointType := (Pos:=(X:=300, Y:=0, Z:=-900));
	PickApproach : McPointType := (Pos:=(X:=-60, Y:=-120, Z:=-800));
	Pick : McPointType := (Pos:=(X:=-60, Y:=-120, Z:=-850));

END_VAR
VAR{AT 'UnloadStat'}
	setUnload : BOOL;
	release : BOOL;
END_VAR
VAR{AT 'UnloadRbt'}
	resetProduct : BOOL;
END_VAR
PROGRAM _MAIN
	Feedrate(100000);
	MoveL(Rest);
	RoundingEdges(50);
	MoveL(PickApproach);
	MoveLR(Pick);
	WaitTime(0.5);
	DO_PATH_SYNCH
		setUnload := TRUE;
		release := TRUE;
	END_PATH_SYNCH
	RoundingEdges(50);
	MoveL(PickApproach);
	MoveL(PlaceApproach);
	MoveL(Place);
	WaitTime(0.5);
	DO_PATH_SYNCH
		resetProduct := TRUE;
	END_PATH_SYNCH
	MoveL(PlaceApproach);
	MoveL(Rest);
END_PROGRAM
```

- Visualisation Logical/mappView (not shown)

Listed in the project but not available here: Logical/Global.typ, Logical/Libraries/AdvIecChk/AdvIecChk.fun, Logical/Source/ShuttleCtrl/ShCtrlGlobalVars.var, Logical/Source/ShuttleCtrl/ShCtrlGlobalTypes.typ, Logical/Source/ShuttleCtrl/ShCtrl/Exit.st, Logical/Source/ProcessStations/ProcGlobalVars.var, Logical/Source/ProcessStations/ProCGlobalTypes.typ, Logical/Source/ProcessStations/FillStation/Exit.st, Logical/Source/ProcessStations/FinishStation/Exit.st, Logical/Source/ProcessStations/FinishStation/LocalFunctionVars.var, Logical/Source/ProcessStations/FinishStation/BatchProcess6DFb.st, Logical/Source/Main/MainGlobalVars.var, Logical/Source/Main/MainGlobalTypes.typ, Logical/Source/Main/Main/Exit.st, Logical/Source/Auxil/AuxGlobalVars.var, Logical/Source/Auxil/AuxGlobalTypes.typ, Logical/Source/Auxil/OeeCalc/Init.st, Logical/Source/Auxil/OeeCalc/Exit.st, Logical/Source/Robots/RobotGlobalVars.var, Logical/Source/Robots/RobotGlobalTypes.typ, Logical/UserPartition/AuditExport
